(* IEC 61131-3 sources: zd/料盘/多料盘, 22 files *)

(* ---- E_料盘运动状态.st ---- *)
{attribute 'qualified_only'}
{attribute 'strict'}
TYPE E_料盘运动状态 :
(

	到取料位中 := 0,
	到放料位中 := 1,
	待机:=4,
	错误:=5,
	暂停:=6,
	手动定位中:=7,
	定位号定位中:=8,
	到初始位中:=9,
	指定取料中:=10,
	指定放料中:=11,
	手动取料中:=12,
	手动放料中:=13
);
END_TYPE

(* ---- S_多料盘管理数据.st ---- *)
TYPE S_多料盘管理数据 :
STRUCT
	料盘管理数据	:ARRAY[0..gvl_常量.最大料盘数量-1] OF S_料盘管理数据;
END_STRUCT
END_TYPE

(* ---- S_多料盘管理数据_HMI.st ---- *)
TYPE S_多料盘管理数据_HMI :
STRUCT
	料盘管理数据索引 :UINT;
	料盘管理数据当前索引 :UINT;
	料盘管理数据	: S_料盘管理数据;
END_STRUCT
END_TYPE

(* ---- S_多料盘管理输入.st ---- *)
TYPE S_多料盘管理输入 :
STRUCT
	手自动:BOOL;

	暂停	:BOOL;
	复位	:BOOL;
	急停	:BOOL;
	报警清除:BOOL;
	//料盘管理输入	:ARRAY[0..gvl_常量.最大料盘数量-1] OF S_料盘管理输入;

	料盘选择	:UINT;
	目标点位 : S_点位行列坐标;                // 目标点位坐标

	设置料盘为满料 : BOOL;
	设置料盘为空料 : BOOL;
	设置点位状态信号 : BOOL;              // 设置点位状态信号
	设置状态 : E_点位状态;                // 设置的状态值

    取料 : BOOL;
	放料 : BOOL;

    定位:BOOL;
    定位号:UINT;

	到初始位:BOOL;

	取料完成:BOOL;
	放料完成:BOOL;
END_STRUCT
END_TYPE

(* ---- S_多料盘管理输入HMI.st ---- *)
TYPE S_多料盘管理输入HMI :
STRUCT

	急停	:BOOL;
	报警清除:BOOL;
	料盘选择	:UINT;
	目标点位 : S_点位行列坐标;                // 目标点位坐标

	设置料盘为满料 : BOOL;
	设置料盘为空料 : BOOL;
	定位到点位信号 : BOOL;
	设置点位状态信号 : BOOL;              // 设置点位状态信号
	设置状态 : E_点位状态;                // 设置的状态值
	定位:BOOL;
    定位号:INT;
	到初始位:BOOL;
END_STRUCT
END_TYPE

(* ---- S_多料盘管理输入HMI_xg_V1.st ---- *)
TYPE S_多料盘管理输入HMI_xg_V1 :
STRUCT

	指定取料	:BOOL;
	指定放料	:BOOL;
	取料	:BOOL;
	放料	:BOOL;

END_STRUCT
END_TYPE

(* ---- S_多料盘管理输出.st ---- *)
TYPE S_多料盘管理输出 :
STRUCT
	定位号定位到位:ARRAY[0..4] OF BOOL;

	初始位定位到位:BOOL;

	占位:DINT;

	到达定位位置:BOOL;

	复位完成:BOOL;
	暂停完成:BOOL;
	料盘运动状态:INT;

    (* 控制输出 *)
    移动X轴信号 : BOOL;                   // X轴移动控制信号
    移动Y轴信号 : BOOL;                   // Y轴移动控制信号
	移动Z轴信号 : BOOL;                   // Z轴移动控制信号
    目标X位置 : REAL;                     // 目标X坐标
    目标Y位置 : REAL;                     // 目标Y坐标
	目标Z位置 : REAL;                     // 目标Z坐标

	当前X位置 : REAL;                     // 目标X坐标
    当前Y位置 : REAL;                     // 目标Y坐标
	当前Z位置 : REAL;                     // 目标Z坐标

	当前X速度 : REAL;                     // 目标X坐标
    当前Y速度 : REAL;                     // 目标Y坐标
	当前Z速度 : REAL;                     // 目标Z坐标

    (* 错误信息 *)
	错误:BOOL;
    错误代码 : E_错误码;
    错误信息 : STRING(100);               // 错误描述

	料盘管理输出	:ARRAY[0..gvl_常量.最大料盘数量-1] OF S_料盘管理输出;
END_STRUCT
END_TYPE

(* ---- S_多料盘管理配置.st ---- *)
TYPE S_多料盘管理配置 :
STRUCT
	x索引	:INT:=0;
	y索引	:INT:=1;
	z索引	:INT:=2;

	x速度:REAL:=50;
	x加速度:REAL:=500;
	x减速度:REAL:=500;

	y速度:REAL:=50;
	y加速度:REAL:=500;
	y减速度:REAL:=500;

// 	xy插补速度:REAL:=50;
// 	xy插补加速度:REAL:=500;
// 	xy插补减速度:REAL:=500;

	z速度:REAL:=50;
	z加速度:REAL:=500;
	z减速度:REAL:=500;

	x定位位置	:ARRAY[0..gvl_常量.最大料盘位置号数量-1] OF REAL:=[10];
	y定位位置	:ARRAY[0..gvl_常量.最大料盘位置号数量-1] OF REAL:=[10];
	z定位位置	:ARRAY[0..gvl_常量.最大料盘位置号数量-1] OF REAL:=[10];

	x轴待料位	:REAL:=10;
	y轴待料位	:REAL:=10;
	z轴待料位	:REAL:=10;

END_STRUCT
END_TYPE

(* ---- S_多料盘管理配置_HMI.st ---- *)
TYPE S_多料盘管理配置_HMI :
STRUCT

	多料盘管理配置: S_多料盘管理配置;
	料盘配置索引:UINT;
	当前料盘配置索引:UINT;

	占位1:REAL;
	占位2:REAL;
	占位3:REAL;
	占位4:REAL;
	占位5:REAL;
	占位6:REAL;
	料盘配置	: S_料盘配置;

	占位14:REAL;
	占位15:REAL;
	占位16:REAL;
	料盘工艺配置:  S_料盘工艺配置;

	多料盘工艺配置:S_多料盘工艺配置;

END_STRUCT
END_TYPE

(* ---- FC_SEL.st ---- *)
//G：BOOL 类型选择条件
//IN0：G = TRUE 时的返回值
//IN1：G = false 时的返回值

FUNCTION FC_SEL : int
VAR_INPUT
	G:BOOL;
	IN1:INT;
	IN2:INT;
END_VAR
VAR
END_VAR

// --- BEGIN IMPLEMENTATION ---

IF G=TRUE THEN
	FC_SEL:=IN1;
	RETURN;
ELSE
	FC_SEL:=IN2;
	RETURN;
END_IF

(* ---- FC_方向判断.st ---- *)
FUNCTION FC_方向判断 : INT
VAR_IN_OUT
	i方向X      : INT;
    i方向Y      : INT;
END_VAR
VAR_INPUT
	f起始点X     : REAL;
    f起始点Y     : REAL;
    f参考点X    : REAL;
    f参考点Y    : REAL;
END_VAR
VAR
	f间距X     : REAL;
    f间距Y     : REAL;
END_VAR

// --- BEGIN IMPLEMENTATION ---

i方向X :=0;
i方向Y :=0;
// 参考点和起始点不能相同
IF f参考点X =f起始点X OR f参考点Y = f起始点Y THEN
	FC_方向判断 := 1;   // 参参考点和起始点不能相同
	RETURN;
END_IF;

// 计算实际与理论的差值
f间距X := f参考点X - f起始点X;
f间距Y := f参考点Y - f起始点Y;

// 判断X方向
i方向X := FC_SEL(f间距X > 0.0, 1, -1);

// 判断Y方向
i方向Y := FC_SEL(f间距Y > 0.0, 1, -1);

(* ---- FB_多料盘管理.st ---- *)
FUNCTION_BLOCK FB_多料盘管理
VAR_IN_OUT
	x轴:SM3_Basic.AXIS_REF_VIRTUAL_SM3;
	y轴:SM3_Basic.AXIS_REF_VIRTUAL_SM3;
	z轴:SM3_Basic.AXIS_REF_VIRTUAL_SM3;

	多料盘管理数据:S_多料盘管理数据;
	多料盘管理输出:S_多料盘管理输出;
	ST_料盘配置V1_xg_0:ARRAY[0..gvl_常量.最大料盘数量-1] OF ST_料盘配置V1_xg;

END_VAR
VAR_INPUT
	全局状态:E_系统运行状态;
	使能:BOOL;
	多料盘管理输入HMI:S_多料盘管理输入HMI;
	S_多料盘管理输入HMI_xg_V1_0:S_多料盘管理输入HMI_xg_V1;
	多料盘管理输入	:S_多料盘管理输入;

	x轴配置:Ax_配置;
	y轴配置:Ax_配置;
	z轴配置:Ax_配置;
	x轴输出:Basic_Lib.Ax_输出;
	y轴输出:Basic_Lib.Ax_输出;
	z轴输出:Basic_Lib.Ax_输出;

	多料盘管理配置:S_多料盘管理配置;
	料盘配置	:ARRAY[0..gvl_常量.最大料盘数量-1] OF S_料盘配置;
	料盘工艺配置	:ARRAY[0..gvl_常量.最大料盘数量-1] OF S_料盘工艺配置;
	多料盘工艺配置	: S_多料盘工艺配置;
	//料盘轴运动输出:S_料盘轴运动输出;
END_VAR
VAR_OUTPUT
	料盘轴运动输入:S_料盘轴运动输入;
	料盘轴运动输出:S_料盘轴运动输出;
	报错料盘:INT;
END_VAR
VAR
	CheckID:Basic_Lib.FB_CheckID;
	//FB_G代码插补_0:FB_G代码插补;
	MC_MoveAbsolute_0: MC_MoveAbsolute;
	MC_MoveAbsolute_1: MC_MoveAbsolute;
	MC_MoveAbsolute_2: MC_MoveAbsolute;
	MC_Move_ChangePosVel_Pul_2: Basic_Lib.MC_Move_ChangePosVel_Pul;
	MC_Stop_1: MC_Stop;
	MC_Stop_2: MC_Stop;
	MC_Stop_3: MC_Stop;
	MC_Reset_0:MC_Reset;
	MC_Reset_1:MC_Reset;
	MC_Reset_2:MC_Reset;

	x轴状态:MC_ReadStatus;
	y轴状态:MC_ReadStatus;
	z轴状态:MC_ReadStatus;
	SMC3_ReinitDrive_0:SMC3_ReinitDrive;
	SMC3_ReinitDrive_1:SMC3_ReinitDrive;
	SMC3_ReinitDrive_2:SMC3_ReinitDrive;

	清空多料盘管理输出:S_多料盘管理输出;

	使能上升沿:R_TRIG;
	设置料盘满料上升沿 :  R_TRIG;  // 设置料盘满料上升沿
	设置料盘空料上升沿 :  R_TRIG;  // 设置料盘空料上升沿
	急停上升沿:  R_TRIG;

	取料上升沿 :  R_TRIG;  // 设置料盘满料上升沿
	放料上升沿 :  R_TRIG;  // 设置料盘空料上升沿
	定位上升沿 :  Standard.R_TRIG;
	到初始位上升沿:Standard.R_TRIG;

	取料完成上升沿 :  R_TRIG;
	放料完成上升沿 :  R_TRIG;
	错误上升沿:R_TRIG;

	手动设置点位状态上升沿:  R_TRIG;
	手动定位点位上升沿:  R_TRIG;
	手动急停上升沿:  R_TRIG;
	手动定位上升沿 :  Standard.R_TRIG;

	手动指定取料上升沿:  R_TRIG;
	手动指定放料上升沿:  R_TRIG;
	手动取料上升沿:  R_TRIG;
	手动放料上升沿:  R_TRIG;

	暂停上升沿:  R_TRIG;
	复位上升沿:  R_TRIG;

	i: INT;
	row: INT;
	col: INT;
	取料流程: INT;
	j: INT;
	临时定位行号: INT;
	临时定位列号: INT;

	z轴定位到位:BOOL;
	放料流程: INT;
	手动定位流程: INT;
	插补定位完成: BOOL;

	定位流程: INT;
	手动定位流程1: INT;

	手动x目标位置:REAL;
	手动y目标位置:REAL;
	手动z目标位置:REAL;

	指定x目标位置:REAL;
	指定y目标位置:REAL;
	指定z目标位置:REAL;

	z轴在待料位:BOOL;

	x轴定位到位: BOOL;
	y轴定位到位: BOOL;
	流程运行状态: BOOL;
	动作控制变量状态: BOOL;
	流程可运行: BOOL;
	轴可运动: BOOL;
	料盘管理输入: INT;
	暂停取料流程: INT;
	暂停定位流程: INT;
	错误前取料流程: INT;
	错误前放料流程: INT;
	错误前定位流程: INT;

	x取料方向X:INT;
	x取料方向Y:INT;
	x放料方向X:INT;
	x放料方向Y:INT;

	i行起始:INT;
	i行结束:INT;
	i列起始:INT;
	i列结束:INT;
	i行递增:INT;
	i列递增:INT;
	指定取料流程: INT;
	指定放料流程: INT;
	手动料盘选择:INT;
	手动取料流程: INT;
	手动放料流程: INT;
END_VAR

// --- BEGIN IMPLEMENTATION ---

(*========================输入控制========================*)
CheckID(xID检测:= TRUE, xID正确=> );
//IF NOT CheckID.xID正确 THEN RETURN; END_IF

IF ADR(x轴) = SM3_Basic.NULL THEN
    RETURN;
END_IF
IF ADR(y轴) = SM3_Basic.NULL  THEN
    RETURN;
END_IF
IF ADR(z轴) = SM3_Basic.NULL  THEN
    RETURN;
END_IF

使能上升沿(CLK:=使能 , Q=> );
IF NOT 使能 THEN
	放料流程:=0;
	取料流程:=0;
	定位流程:=0;
	手动定位流程:=0;
	指定取料流程:=0;
	指定放料流程:=0;
	手动取料流程:=0;
	手动放料流程:=0;
	多料盘管理输出.料盘运动状态:=E_料盘运动状态.待机;
	料盘轴运动输入.x轴定位:=FALSE;
	料盘轴运动输入.y轴定位:=FALSE;
	料盘轴运动输入.Z轴定位:=FALSE;
	料盘轴运动输入.插补启动:=FALSE;
	多料盘管理输出.错误:=FALSE;
	多料盘管理输出.错误信息:='';
	RETURN;
ELSE
	;
END_IF

ACT_自动状态控制();

设置料盘满料上升沿(CLK := (多料盘管理输入.设置料盘为满料  AND 多料盘管理输入.手自动) OR (多料盘管理输入HMI.设置料盘为满料  AND NOT 多料盘管理输入.手自动));
设置料盘空料上升沿(CLK := (多料盘管理输入.设置料盘为空料 AND 多料盘管理输入.手自动) OR (多料盘管理输入HMI.设置料盘为空料  AND NOT 多料盘管理输入.手自动));
(* 处理料盘设置满料信号 *)
IF 设置料盘满料上升沿.Q THEN
	(* 初始化指定料盘数据 *)
	FOR row := 0 TO GVL_常量.最大料盘行数 - 1 DO
		FOR col := 0 TO GVL_常量.最大料盘列数 - 1 DO
			IF 多料盘管理输入.料盘选择<=GVL_常量.最大料盘数量-1 THEN
				IF  多料盘管理输入.手自动 THEN
					多料盘管理数据.料盘管理数据[多料盘管理输入.料盘选择].点位状态[row, col] := E_点位状态.有料;
					多料盘管理数据.料盘管理数据[多料盘管理输入.料盘选择].屏蔽点位[row, col] := FALSE;
				ELSE
					多料盘管理数据.料盘管理数据[多料盘管理输入HMI.料盘选择].点位状态[row, col] := E_点位状态.有料;
					多料盘管理数据.料盘管理数据[多料盘管理输入HMI.料盘选择].屏蔽点位[row, col] := FALSE;
				END_IF

			END_IF

		END_FOR;
	END_FOR;
	IF 多料盘管理输入.料盘选择>GVL_常量.最大料盘数量-1 THEN
	FOR i := 0 TO GVL_常量.最大料盘数量 - 1 DO
		FOR row := 0 TO GVL_常量.最大料盘行数 - 1 DO
			FOR col := 0 TO GVL_常量.最大料盘列数 - 1 DO

				多料盘管理数据.料盘管理数据[i].点位状态[row, col] := E_点位状态.有料;
				多料盘管理数据.料盘管理数据[i].屏蔽点位[row, col] := FALSE;

			END_FOR;
		END_FOR;
	END_FOR
	END_IF
END_IF;

(* 处理料盘设置空料信号 *)
IF 设置料盘空料上升沿.Q THEN
	(* 初始化指定料盘数据 *)
	FOR row := 0 TO GVL_常量.最大料盘行数 - 1 DO
		FOR col := 0 TO GVL_常量.最大料盘列数 - 1 DO
			IF 多料盘管理输入.料盘选择<=GVL_常量.最大料盘数量-1 THEN
				IF  多料盘管理输入.手自动 THEN
					多料盘管理数据.料盘管理数据[多料盘管理输入.料盘选择].点位状态[row, col] := E_点位状态.无料;
					多料盘管理数据.料盘管理数据[多料盘管理输入.料盘选择].屏蔽点位[row, col] := FALSE;
				ELSE
					多料盘管理数据.料盘管理数据[多料盘管理输入HMI.料盘选择].点位状态[row, col] := E_点位状态.无料;
					多料盘管理数据.料盘管理数据[多料盘管理输入HMI.料盘选择].屏蔽点位[row, col] := FALSE;
				END_IF
			END_IF
		END_FOR;

		IF 多料盘管理输入.料盘选择>GVL_常量.最大料盘数量-1 THEN
		FOR i := 0 TO GVL_常量.最大料盘数量 - 1 DO
			FOR row := 0 TO GVL_常量.最大料盘行数 - 1 DO
				FOR col := 0 TO GVL_常量.最大料盘列数 - 1 DO

					多料盘管理数据.料盘管理数据[i].点位状态[row, col] := E_点位状态.无料;
					多料盘管理数据.料盘管理数据[i].屏蔽点位[row, col] := FALSE;

				END_FOR;
			END_FOR;
		END_FOR
		END_IF
	END_FOR;
END_IF;

手动设置点位状态上升沿(CLK:=多料盘管理输入HMI.设置点位状态信号 , Q=> );
IF 手动设置点位状态上升沿.Q AND ((多料盘管理输入HMI.目标点位.行号<>临时定位行号 OR 多料盘管理输入HMI.目标点位.列号<>临时定位列号)OR (放料流程=0 AND 取料流程=0))  THEN
	多料盘管理数据.料盘管理数据[多料盘管理输入HMI.料盘选择].点位状态[多料盘管理输入HMI.目标点位.行号,多料盘管理输入HMI.目标点位.列号]:=多料盘管理输入HMI.设置状态;
	多料盘管理数据.料盘管理数据[多料盘管理输入HMI.料盘选择].屏蔽点位[多料盘管理输入HMI.目标点位.行号,多料盘管理输入HMI.目标点位.列号]:=(多料盘管理输入HMI.设置状态=E_点位状态.屏蔽);
END_IF

流程可运行:=放料流程=0 AND 取料流程=0 AND 定位流程=0 AND 手动定位流程=0 AND 指定取料流程=0 AND 指定放料流程=0 AND 手动取料流程=0 AND 手动放料流程=0 ;

轴可运动:= x轴状态.Standstill AND y轴状态.Standstill AND z轴状态.Standstill ;
//x轴输出.x回零完成 AND y轴输出.x回零完成 AND z轴输出.x回零完成  AND

ACT_手动();
ACT_手动指定放料();
ACT_手动指定取料();
ACT_手动放料();
ACT_手动取料();
ACT_自动取料();
ACT_自动放料();
ACT_定位号插补();

ACT_FB();

多料盘管理输出.初始位定位到位:=(x轴.fActPosition<=(多料盘管理配置.x轴待料位+x轴配置.f到位偏差)) AND (x轴.fActPosition>=(多料盘管理配置.x轴待料位-x轴配置.f到位偏差))
	AND(y轴.fActPosition<=(多料盘管理配置.y轴待料位+y轴配置.f到位偏差)) AND (y轴.fActPosition>=(多料盘管理配置.y轴待料位-y轴配置.f到位偏差))
	AND (z轴.fActPosition<=(多料盘管理配置.z轴待料位+z轴配置.f到位偏差)) AND (z轴.fActPosition>=(多料盘管理配置.z轴待料位-z轴配置.f到位偏差)
	AND  x轴状态.Standstill AND y轴状态.Standstill AND z轴状态.Standstill );

插补定位完成:=((x轴.fActPosition<=(料盘轴运动输入.目标位置[0]+x轴配置.f到位偏差)) AND (x轴.fActPosition>=(料盘轴运动输入.目标位置[0]-x轴配置.f到位偏差))
AND(y轴.fActPosition<=(料盘轴运动输入.目标位置[1]+y轴配置.f到位偏差)) AND (y轴.fActPosition>=(料盘轴运动输入.目标位置[1]-y轴配置.f到位偏差)));

x轴定位到位:=((x轴.fActPosition<=(料盘轴运动输入.x定位位置+x轴配置.f到位偏差)) AND (x轴.fActPosition>=(料盘轴运动输入.x定位位置-x轴配置.f到位偏差)));
y轴定位到位:=((y轴.fActPosition<=(料盘轴运动输入.y定位位置+y轴配置.f到位偏差)) AND (y轴.fActPosition>=(料盘轴运动输入.y定位位置-y轴配置.f到位偏差)));
z轴定位到位:=((z轴.fActPosition<=(料盘轴运动输入.z定位位置+z轴配置.f到位偏差)) AND (z轴.fActPosition>=(料盘轴运动输入.z定位位置-z轴配置.f到位偏差)));

z轴在待料位:=(z轴.fActPosition<=(多料盘管理配置.z轴待料位+z轴配置.f到位偏差)) AND (z轴.fActPosition>=(多料盘管理配置.z轴待料位-z轴配置.f到位偏差));

ACT_料盘状态();

//手自动报警清除
IF 多料盘管理输入.报警清除 OR 多料盘管理输入hmi.报警清除 THEN
	多料盘管理输出.错误:=FALSE;
    多料盘管理输出.错误信息 :='';              // 系统错误描述
	//多料盘管理输出.料盘运动状态:=E_料盘运动状态.待机;
END_IF

IF 料盘轴运动输出.x定位错误 THEN 多料盘管理输出.错误:=TRUE; 多料盘管理输出.错误信息 := Standard.CONCAT('SMC_ERROR: ', TO_STRING(料盘轴运动输出.x定位错误码));多料盘管理输出.错误代码:=E_错误码.料盘X轴定位错误; END_IF
IF 料盘轴运动输出.y定位错误 THEN 多料盘管理输出.错误:=TRUE; 多料盘管理输出.错误信息 := Standard.CONCAT('SMC_ERROR: ', TO_STRING(料盘轴运动输出.y定位错误码));多料盘管理输出.错误代码:=E_错误码.料盘Y轴定位错误; END_IF
IF 料盘轴运动输出.z定位错误 THEN 多料盘管理输出.错误:=TRUE; 多料盘管理输出.错误信息 :=MC_Move_ChangePosVel_Pul_2.s错误码; (*Standard.CONCAT('SMC_ERROR: ', TO_STRING(料盘轴运动输出.z定位错误码));*)多料盘管理输出.错误代码:=E_错误码.料盘Z轴定位错误; END_IF
//IF LS_2AxisLine_1.Error  THEN 多料盘管理输出.错误:=TRUE; 多料盘管理输出.错误信息 := Standard.CONCAT('SMC_ERROR: ', TO_STRING(LS_2AxisLine_1.ErrorID)); 多料盘管理输出.错误代码:=3; END_IF
//IF 料盘轴运动输出.插补错误 THEN 多料盘管理输出.错误:=TRUE; 多料盘管理输出.错误信息 := 料盘轴运动输出.插补错误码;多料盘管理输出.错误代码:=3; END_IF

错误上升沿(CLK:= 多料盘管理输出.错误, Q=> );
IF 错误上升沿.Q THEN
	;
	放料流程:=0;
	取料流程:=0;
	定位流程:=0;
	手动定位流程:=0;
	指定取料流程:=0;
	指定放料流程:=0;
	手动取料流程:=0;
	手动放料流程:=0;
	料盘轴运动输入.x轴定位:=FALSE;
	料盘轴运动输入.y轴定位:=FALSE;
	料盘轴运动输入.Z轴定位:=FALSE;
	料盘轴运动输入.插补启动:=FALSE;
	多料盘管理输出.料盘运动状态:=E_料盘运动状态.错误;
END_IF

IF 多料盘管理输出.错误 THEN
	;
	放料流程:=0;
	取料流程:=0;
	定位流程:=0;
	手动定位流程:=0;
	指定取料流程:=0;
	手动取料流程:=0;
	手动放料流程:=0;
	料盘轴运动输入.x轴定位:=FALSE;
	料盘轴运动输入.y轴定位:=FALSE;
	料盘轴运动输入.Z轴定位:=FALSE;
	料盘轴运动输入.插补启动:=FALSE;
END_IF

(* ---- FB_多料盘管理.ACT_定位号插补.action.st ---- *)
定位上升沿(CLK:=多料盘管理输入.定位 AND 多料盘管理输入.手自动 , Q=> );

IF GVL_系统变量.全局状态=E_系统运行状态.系统状态_故障 THEN
	料盘轴运动输入.x轴定位:=FALSE;
	料盘轴运动输入.y轴定位:=FALSE;
	料盘轴运动输入.Z轴定位:=FALSE;
	料盘轴运动输入.插补启动:=FALSE;
	RETURN;
END_IF

IF GVL_系统变量.全局状态<>E_系统运行状态.系统状态_运行 AND GVL_系统变量.全局状态<>E_系统运行状态.系统状态_清料中  AND GVL_系统变量.全局状态<>E_系统运行状态.系统状态_暂停中 THEN

	RETURN;
END_IF
IF 定位上升沿.Q AND 轴可运动 AND 流程可运行
	AND NOT 多料盘管理输入.到初始位 AND NOT 多料盘管理输入.取料 AND NOT 多料盘管理输入.放料
	 AND NOT 多料盘管理输入.暂停 AND NOT 多料盘管理输出.错误
	AND 多料盘管理输入.定位号>=0 AND 多料盘管理输入.定位号<5 AND

	(多料盘管理输出.料盘运动状态=E_料盘运动状态.待机
	OR 多料盘管理输出.料盘运动状态=E_料盘运动状态.暂停)
THEN

		料盘轴运动输入.x轴定位:=FALSE;
		料盘轴运动输入.y轴定位:=FALSE;
		料盘轴运动输入.Z轴定位:=FALSE;
		料盘轴运动输入.插补启动:=FALSE;
		多料盘管理输出.定位号定位到位[多料盘管理输入.定位号]:=FALSE;
		多料盘管理输出.料盘运动状态:=E_料盘运动状态.定位号定位中;
		定位流程:=2;

ELSE
	;
END_IF;

IF 定位流程=2 THEN
	IF z轴在待料位=FALSE AND NOT 多料盘管理输入.暂停 THEN
		料盘轴运动输入.z定位位置:=多料盘管理输出.目标Z位置 := 多料盘管理配置.z轴待料位;
		料盘轴运动输入.z定位速度:=多料盘管理配置.z速度;
		料盘轴运动输入.z定位加速度:=多料盘管理配置.z加速度;
		料盘轴运动输入.z定位减速度:=多料盘管理配置.z减速度;
		(* 移动轴 *)
		多料盘管理输出.移动Z轴信号 := TRUE;
		料盘轴运动输入.Z轴定位:=TRUE;
	ELSIF z轴在待料位 AND NOT 多料盘管理输入.暂停 THEN
		多料盘管理输出.移动Z轴信号 := FALSE;
		料盘轴运动输入.Z轴定位:=FALSE;
		定位流程:=5;
	ELSIF  多料盘管理输入.暂停 THEN
		多料盘管理输出.暂停完成:=TRUE;
	END_IF
END_IF

IF 定位流程=5 THEN

		多料盘管理输出.移动X轴信号 := FALSE;
		多料盘管理输出.移动Y轴信号 := FALSE;

		//料盘轴运动输入.插补启动:=FALSE;

		料盘轴运动输入.x轴定位:=FALSE;
		料盘轴运动输入.y轴定位:=FALSE;
		料盘轴运动输入.x定位位置:=料盘轴运动输入.目标位置[0] :=多料盘管理输出.目标X位置 := 多料盘管理配置.x定位位置[多料盘管理输入.定位号];

		料盘轴运动输入.y定位位置:=料盘轴运动输入.目标位置[1] :=多料盘管理输出.目标Y位置 := 多料盘管理配置.y定位位置[多料盘管理输入.定位号];

		料盘轴运动输入.z定位位置:=多料盘管理输出.目标Z位置 := 多料盘管理配置.z定位位置[多料盘管理输入.定位号];
		// 		料盘轴运动输入.xy插补速度:=多料盘管理配置.xy插补速度;
		// 		料盘轴运动输入.xy插补加速度:=多料盘管理配置.xy插补加速度;
		// 		料盘轴运动输入.xy插补减速度:=多料盘管理配置.xy插补减速度;
		料盘轴运动输入.x定位速度:=多料盘管理配置.x速度;
		料盘轴运动输入.x定位加速度:=多料盘管理配置.x加速度;
		料盘轴运动输入.x定位减速度:=多料盘管理配置.x减速度;

		料盘轴运动输入.y定位速度:=多料盘管理配置.y速度;
		料盘轴运动输入.y定位加速度:=多料盘管理配置.y加速度;
		料盘轴运动输入.y定位减速度:=多料盘管理配置.y减速度;

		IF 多料盘工艺配置.位置号z轴下降减速[多料盘管理输入.定位号].启用=1 THEN
			IF z轴.fActPosition>多料盘工艺配置.位置号z轴下降减速[多料盘管理输入.定位号].z定位减速位置 THEN
				料盘轴运动输入.z定位速度:= 多料盘工艺配置.位置号z轴下降减速[多料盘管理输入.定位号].z定位减速速度;
			ELSE
				料盘轴运动输入.z定位速度:=多料盘管理配置.z速度;
			END_IF
		ELSE
			料盘轴运动输入.z定位速度:=多料盘管理配置.z速度;
		END_IF
		料盘轴运动输入.z定位速度:=多料盘管理配置.z速度;
		料盘轴运动输入.z定位加速度:=多料盘管理配置.z加速度;
		料盘轴运动输入.z定位减速度:=多料盘管理配置.z减速度;

		定位流程:=10;

ELSIF 定位流程=10 THEN

	(* 移动轴 *)

	IF 插补定位完成=FALSE AND x轴.nAxisState=Standstill  AND y轴.nAxisState=Standstill AND NOT 多料盘管理输入.暂停 THEN
		多料盘管理输出.移动X轴信号 := TRUE;
		多料盘管理输出.移动Y轴信号 := TRUE;
		//料盘轴运动输入.插补启动:=TRUE;
		料盘轴运动输入.x轴定位:=TRUE;
		料盘轴运动输入.y轴定位:=TRUE;
	ELSIF 插补定位完成 AND x轴.nAxisState=Standstill  AND y轴.nAxisState=Standstill AND NOT 多料盘管理输入.暂停 THEN
		多料盘管理输出.移动X轴信号 := FALSE;
		多料盘管理输出.移动Y轴信号 := FALSE;

		//料盘轴运动输入.插补启动:=FALSE;

		料盘轴运动输入.x轴定位:=FALSE;
		料盘轴运动输入.y轴定位:=FALSE;
		定位流程:=12;
	ELSIF  多料盘管理输入.暂停 THEN
		多料盘管理输出.暂停完成:=TRUE;
	END_IF
ELSIF 定位流程=12 THEN

		IF 多料盘工艺配置.位置号z轴下降减速[多料盘管理输入.定位号].启用=1 THEN
			IF z轴.fActPosition>多料盘工艺配置.位置号z轴下降减速[多料盘管理输入.定位号].z定位减速位置 THEN
				料盘轴运动输入.z定位速度:= 多料盘工艺配置.位置号z轴下降减速[多料盘管理输入.定位号].z定位减速速度;
			END_IF
		END_IF
		IF z轴定位到位=FALSE AND  z轴.nAxisState=Standstill  AND NOT 多料盘管理输入.暂停 THEN
			(* 移动轴 *)
			多料盘管理输出.移动Z轴信号 := TRUE;
			料盘轴运动输入.Z轴定位:=TRUE;
		ELSIF z轴定位到位 AND z轴.nAxisState=Standstill AND NOT 多料盘管理输入.暂停 THEN
			多料盘管理输出.移动Z轴信号 := FALSE;
			料盘轴运动输入.Z轴定位:=FALSE;
			定位流程:=13;
		ELSIF z轴定位到位 AND 多料盘管理输入.暂停 THEN
			多料盘管理输出.暂停完成:=TRUE;
		END_IF

END_IF

IF 定位流程=13 THEN

		IF 多料盘管理输出.料盘运动状态=E_料盘运动状态.定位号定位中 THEN
			IF 多料盘工艺配置.位置号附加动作[多料盘管理输入.定位号].位置号附加动作=0 THEN
				多料盘管理输出.料盘运动状态:=E_料盘运动状态.待机;
				多料盘管理输出.定位号定位到位[多料盘管理输入.定位号]:=TRUE;
				定位流程:=0;
			ELSIF 多料盘工艺配置.位置号附加动作[多料盘管理输入.定位号].位置号附加动作=1 THEN
				定位流程:=20;
			END_IF
		ELSE
			多料盘管理输出.料盘运动状态:=E_料盘运动状态.待机;
			定位流程:=0;
		END_IF

ELSIF 定位流程=20 THEN
	IF 多料盘工艺配置.位置号附加动作[多料盘管理输入.定位号].索引=0 AND x轴.nAxisState=Standstill AND NOT 多料盘管理输入.暂停 THEN
		料盘轴运动输入.X定位位置:=多料盘管理输出.目标X位置 := 多料盘工艺配置.位置号附加动作[多料盘管理输入.定位号].偏移值+x轴.fActPosition;
		料盘轴运动输入.x定位速度:= 多料盘工艺配置.位置号附加动作[多料盘管理输入.定位号].速度;
		料盘轴运动输入.x定位加速度:= 多料盘工艺配置.位置号附加动作[多料盘管理输入.定位号].加速度;
		料盘轴运动输入.x定位减速度:=多料盘工艺配置.位置号附加动作[多料盘管理输入.定位号].减速度;
		多料盘管理输出.移动X轴信号 := TRUE;
		料盘轴运动输入.x轴定位:=TRUE;
		定位流程:=30;
	ELSIF 多料盘工艺配置.位置号附加动作[多料盘管理输入.定位号].索引=1 AND y轴.nAxisState=Standstill AND NOT 多料盘管理输入.暂停 THEN
		料盘轴运动输入.y定位位置:=多料盘管理输出.目标y位置 := 多料盘工艺配置.位置号附加动作[多料盘管理输入.定位号].偏移值+y轴.fActPosition;
		料盘轴运动输入.y定位速度:=多料盘工艺配置.位置号附加动作[多料盘管理输入.定位号].速度;
		料盘轴运动输入.y定位加速度:=多料盘工艺配置.位置号附加动作[多料盘管理输入.定位号].加速度;
		料盘轴运动输入.y定位减速度:=多料盘工艺配置.位置号附加动作[多料盘管理输入.定位号].减速度;
		多料盘管理输出.移动y轴信号 := TRUE;
		料盘轴运动输入.y轴定位:=TRUE;
		定位流程:=30;
	ELSIF 多料盘工艺配置.位置号附加动作[多料盘管理输入.定位号].索引=2 AND z轴.nAxisState=Standstill AND NOT 多料盘管理输入.暂停 THEN
		料盘轴运动输入.z定位位置:=多料盘管理输出.目标z位置 := 多料盘工艺配置.位置号附加动作[多料盘管理输入.定位号].偏移值+z轴.fActPosition;
		料盘轴运动输入.z定位速度:=多料盘工艺配置.位置号附加动作[多料盘管理输入.定位号].速度;
		料盘轴运动输入.z定位加速度:=多料盘工艺配置.位置号附加动作[多料盘管理输入.定位号].加速度;
		料盘轴运动输入.z定位减速度:=多料盘工艺配置.位置号附加动作[多料盘管理输入.定位号].减速度;
		多料盘管理输出.移动z轴信号 := TRUE;
		料盘轴运动输入.z轴定位:=TRUE;
		定位流程:=30;
	ELSIF 多料盘管理输入.暂停 THEN
		多料盘管理输出.暂停完成:=TRUE;
	END_IF

ELSIF 定位流程=30 THEN
	IF 多料盘工艺配置.位置号附加动作[多料盘管理输入.定位号].索引=0 THEN
		IF x轴定位到位 AND x轴.nAxisState=Standstill THEN
			料盘轴运动输入.x轴定位:=FALSE;
			多料盘管理输出.移动X轴信号 := FALSE;
			多料盘管理输出.料盘运动状态:=E_料盘运动状态.待机;
			多料盘管理输出.定位号定位到位[多料盘管理输入.定位号]:=TRUE;
			定位流程:=0;
		END_IF
	ELSIF 多料盘工艺配置.位置号附加动作[多料盘管理输入.定位号].索引=1 THEN
		IF y轴定位到位 AND y轴.nAxisState=Standstill THEN
			料盘轴运动输入.y轴定位:=FALSE;
			多料盘管理输出.移动y轴信号 := FALSE;
			多料盘管理输出.料盘运动状态:=E_料盘运动状态.待机;
			多料盘管理输出.定位号定位到位[多料盘管理输入.定位号]:=TRUE;
			定位流程:=0;
		END_IF
	ELSIF 多料盘工艺配置.位置号附加动作[多料盘管理输入.定位号].索引=2 THEN
		IF z轴定位到位 AND z轴.nAxisState=Standstill THEN
			料盘轴运动输入.z轴定位:=FALSE;
			多料盘管理输出.移动z轴信号 := FALSE;
			多料盘管理输出.料盘运动状态:=E_料盘运动状态.待机;
			多料盘管理输出.定位号定位到位[多料盘管理输入.定位号]:=TRUE;
			定位流程:=0;
		END_IF
	END_IF
END_IF

(* ---- FB_多料盘管理.ACT_手动.action.st ---- *)
手动定位上升沿(CLK:=多料盘管理输入HMI.定位 AND NOT 多料盘管理输入.手自动, Q=> );
到初始位上升沿(CLK:=多料盘管理输入HMI.到初始位 AND NOT 多料盘管理输入.手自动  , Q=> );
手动定位点位上升沿(CLK:=多料盘管理输入HMI.定位到点位信号 AND NOT 多料盘管理输入.手自动 , Q=> );

IF 手动定位点位上升沿.Q AND 轴可运动 AND 流程可运行 THEN
	料盘轴运动输入.x轴定位:=FALSE;
	料盘轴运动输入.y轴定位:=FALSE;
	料盘轴运动输入.Z轴定位:=FALSE;
	料盘轴运动输入.插补启动:=FALSE;
	手动定位流程:=2;
	多料盘管理输出.料盘运动状态:=E_料盘运动状态.手动定位中;

END_IF

IF 手动定位上升沿.Q AND 轴可运动 AND 流程可运行  THEN
	料盘轴运动输入.x轴定位:=FALSE;
	料盘轴运动输入.y轴定位:=FALSE;
	料盘轴运动输入.Z轴定位:=FALSE;
	料盘轴运动输入.插补启动:=FALSE;
	多料盘管理输出.定位号定位到位[多料盘管理输入hmi.定位号]:=FALSE;
	手动定位流程:=2;
	多料盘管理输出.料盘运动状态:=E_料盘运动状态.定位号定位中;

END_IF

IF 到初始位上升沿.Q  AND 轴可运动 AND 流程可运行 THEN
	料盘轴运动输入.x轴定位:=FALSE;
	料盘轴运动输入.y轴定位:=FALSE;
	料盘轴运动输入.Z轴定位:=FALSE;
	料盘轴运动输入.插补启动:=FALSE;
	多料盘管理输出.料盘运动状态:=E_料盘运动状态.到初始位中;
	手动定位流程:=2;

ELSE
	;
END_IF;

手动x目标位置:=料盘配置[多料盘管理输入HMI.料盘选择].起始X坐标 +
								多料盘管理输入HMI.目标点位.列号 * 料盘配置[多料盘管理输入HMI.料盘选择].列间距 +
								料盘配置[多料盘管理输入HMI.料盘选择].点位偏移[多料盘管理输入HMI.目标点位.行号, 多料盘管理输入HMI.目标点位.列号].x点位偏移;
手动y目标位置:=	料盘配置[多料盘管理输入HMI.料盘选择].起始Y坐标 +
								多料盘管理输入HMI.目标点位.行号 * 料盘配置[多料盘管理输入HMI.料盘选择].行间距 +
								料盘配置[多料盘管理输入HMI.料盘选择].点位偏移[多料盘管理输入HMI.目标点位.行号, 多料盘管理输入HMI.目标点位.列号].y点位偏移;
手动z目标位置:=料盘配置[多料盘管理输入HMI.料盘选择].Z轴高度 +
								料盘配置[多料盘管理输入HMI.料盘选择].点位偏移[多料盘管理输入HMI.目标点位.行号, 多料盘管理输入HMI.目标点位.列号].z点位偏移;

IF 手动定位流程=2 THEN
	IF z轴在待料位=FALSE THEN
		料盘轴运动输入.z定位位置:=多料盘管理输出.目标Z位置 := 多料盘管理配置.z轴待料位;
		料盘轴运动输入.z定位速度:=多料盘管理配置.z速度;
		料盘轴运动输入.z定位加速度:=多料盘管理配置.z加速度;
		料盘轴运动输入.z定位减速度:=多料盘管理配置.z减速度;
		料盘轴运动输入.Z轴定位:=TRUE;
		手动定位流程:=5;
	ELSE
		手动定位流程:=5;
	END_IF
END_IF

IF 手动定位流程=5 THEN
	IF z轴在待料位 AND z轴.nAxisState=Standstill  THEN
		IF 多料盘管理输出.料盘运动状态=E_料盘运动状态.手动定位中 THEN
			料盘轴运动输入.x定位位置:=料盘轴运动输入.目标位置[0] :=多料盘管理输出.目标X位置 := 料盘配置[多料盘管理输入HMI.料盘选择].起始X坐标 +
									多料盘管理输入HMI.目标点位.列号 * 料盘配置[多料盘管理输入HMI.料盘选择].列间距 +
									料盘配置[多料盘管理输入HMI.料盘选择].点位偏移[多料盘管理输入HMI.目标点位.行号, 多料盘管理输入HMI.目标点位.列号].x点位偏移;

			料盘轴运动输入.y定位位置:=料盘轴运动输入.目标位置[1] :=多料盘管理输出.目标Y位置 := 料盘配置[多料盘管理输入HMI.料盘选择].起始Y坐标 +
										多料盘管理输入HMI.目标点位.行号 * 料盘配置[多料盘管理输入HMI.料盘选择].行间距 +
										料盘配置[多料盘管理输入HMI.料盘选择].点位偏移[多料盘管理输入HMI.目标点位.行号, 多料盘管理输入HMI.目标点位.列号].y点位偏移;

			料盘轴运动输入.z定位位置:=多料盘管理输出.目标Z位置 := 料盘配置[多料盘管理输入HMI.料盘选择].Z轴高度 +
										料盘配置[多料盘管理输入HMI.料盘选择].点位偏移[多料盘管理输入HMI.目标点位.行号, 多料盘管理输入HMI.目标点位.列号].z点位偏移;
		ELSIF 多料盘管理输出.料盘运动状态=E_料盘运动状态.定位号定位中 THEN
			料盘轴运动输入.x定位位置:=料盘轴运动输入.目标位置[0] :=多料盘管理输出.目标X位置 := 多料盘管理配置.x定位位置[多料盘管理输入HMI.定位号];

			料盘轴运动输入.y定位位置:=料盘轴运动输入.目标位置[1] :=多料盘管理输出.目标Y位置 := 多料盘管理配置.y定位位置[多料盘管理输入HMI.定位号];

			料盘轴运动输入.z定位位置:=多料盘管理输出.目标Z位置 := 多料盘管理配置.z定位位置[多料盘管理输入HMI.定位号];
		ELSIF 多料盘管理输出.料盘运动状态=E_料盘运动状态.到初始位中 THEN
			料盘轴运动输入.x定位位置:=料盘轴运动输入.目标位置[0] :=多料盘管理输出.目标X位置 := 多料盘管理配置.x轴待料位;

			料盘轴运动输入.y定位位置:=料盘轴运动输入.目标位置[1] :=多料盘管理输出.目标Y位置 := 多料盘管理配置.y轴待料位;

			料盘轴运动输入.z定位位置:=多料盘管理输出.目标Z位置 := 多料盘管理配置.z轴待料位;
		END_IF
// 		料盘轴运动输入.xy插补速度:=多料盘管理配置.xy插补速度;
// 		料盘轴运动输入.xy插补加速度:=多料盘管理配置.xy插补加速度;
// 		料盘轴运动输入.xy插补减速度:=多料盘管理配置.xy插补减速度;

		料盘轴运动输入.x定位速度:=多料盘管理配置.x速度;
		料盘轴运动输入.x定位加速度:=多料盘管理配置.x加速度;
		料盘轴运动输入.x定位减速度:=多料盘管理配置.x减速度;

		料盘轴运动输入.y定位速度:=多料盘管理配置.y速度;
		料盘轴运动输入.y定位加速度:=多料盘管理配置.y加速度;
		料盘轴运动输入.y定位减速度:=多料盘管理配置.y减速度;

		料盘轴运动输入.z定位速度:=多料盘管理配置.z速度;
		料盘轴运动输入.z定位加速度:=多料盘管理配置.z加速度;
		料盘轴运动输入.z定位减速度:=多料盘管理配置.z减速度;
		料盘轴运动输入.Z轴定位:=FALSE;
		手动定位流程:=10;

	END_IF
END_IF

IF 手动定位流程=10 THEN

	//料盘轴运动输入.插补启动:=TRUE;

	料盘轴运动输入.x轴定位:=TRUE;
	料盘轴运动输入.y轴定位:=TRUE;

	手动定位流程:=12;
ELSIF 手动定位流程=12 THEN
	IF 插补定位完成 AND x轴.nAxisState=Standstill  AND y轴.nAxisState=Standstill  THEN

		//料盘轴运动输入.插补启动:=FALSE;

		料盘轴运动输入.x轴定位:=FALSE;
		料盘轴运动输入.y轴定位:=FALSE;

		IF z轴.nAxisState=Standstill  THEN
			料盘轴运动输入.Z轴定位:=TRUE;
			手动定位流程:=13;
		END_IF

	END_IF
END_IF

IF 手动定位流程=13 THEN
	IF 多料盘管理输出.料盘运动状态=E_料盘运动状态.定位号定位中 THEN
		IF 多料盘工艺配置.位置号z轴下降减速[多料盘管理输入HMI.定位号].启用=1 THEN
			IF z轴.fActPosition>多料盘工艺配置.位置号z轴下降减速[多料盘管理输入HMI.定位号].z定位减速位置 THEN
				料盘轴运动输入.z定位速度:= 多料盘工艺配置.位置号z轴下降减速[多料盘管理输入HMI.定位号].z定位减速速度;		END_IF
		END_IF
	END_IF
	IF z轴定位到位 AND z轴.nAxisState=Standstill  THEN
		料盘轴运动输入.Z轴定位:=FALSE;
		IF 多料盘管理输出.料盘运动状态=E_料盘运动状态.定位号定位中 THEN
			IF 多料盘工艺配置.位置号附加动作[多料盘管理输入hmi.定位号].位置号附加动作=0 THEN
				多料盘管理输出.料盘运动状态:=E_料盘运动状态.待机;
				多料盘管理输出.定位号定位到位[多料盘管理输入hmi.定位号]:=TRUE;
				手动定位流程:=0;
			ELSIF 多料盘工艺配置.位置号附加动作[多料盘管理输入hmi.定位号].位置号附加动作=1 THEN
				手动定位流程:=20;
			END_IF
		ELSE
			多料盘管理输出.料盘运动状态:=E_料盘运动状态.待机;
			手动定位流程:=0;
		END_IF

	END_IF

ELSIF 手动定位流程=20 THEN
	IF 多料盘工艺配置.位置号附加动作[多料盘管理输入hmi.定位号].索引=0 THEN
		料盘轴运动输入.X定位位置:=多料盘管理输出.目标X位置 := 多料盘工艺配置.位置号附加动作[多料盘管理输入hmi.定位号].偏移值+x轴.fActPosition;
		料盘轴运动输入.x定位速度:= 多料盘工艺配置.位置号附加动作[多料盘管理输入hmi.定位号].速度;
		料盘轴运动输入.x定位加速度:= 多料盘工艺配置.位置号附加动作[多料盘管理输入hmi.定位号].加速度;
		料盘轴运动输入.x定位减速度:=多料盘工艺配置.位置号附加动作[多料盘管理输入hmi.定位号].减速度;
		料盘轴运动输入.x轴定位:=TRUE;
		手动定位流程:=30;
	ELSIF 多料盘工艺配置.位置号附加动作[多料盘管理输入hmi.定位号].索引=1 THEN
		料盘轴运动输入.y定位位置:=多料盘管理输出.目标y位置 := 多料盘工艺配置.位置号附加动作[多料盘管理输入hmi.定位号].偏移值+y轴.fActPosition;
		料盘轴运动输入.y定位速度:=多料盘工艺配置.位置号附加动作[多料盘管理输入hmi.定位号].速度;
		料盘轴运动输入.y定位加速度:=多料盘工艺配置.位置号附加动作[多料盘管理输入hmi.定位号].加速度;
		料盘轴运动输入.y定位减速度:=多料盘工艺配置.位置号附加动作[多料盘管理输入hmi.定位号].减速度;
		料盘轴运动输入.y轴定位:=TRUE;
		手动定位流程:=30;
	ELSIF 多料盘工艺配置.位置号附加动作[多料盘管理输入hmi.定位号].索引=2 THEN
		料盘轴运动输入.z定位位置:=多料盘管理输出.目标z位置 := 多料盘工艺配置.位置号附加动作[多料盘管理输入hmi.定位号].偏移值+z轴.fActPosition;
		料盘轴运动输入.z定位速度:=多料盘工艺配置.位置号附加动作[多料盘管理输入hmi.定位号].速度;
		料盘轴运动输入.z定位加速度:=多料盘工艺配置.位置号附加动作[多料盘管理输入hmi.定位号].加速度;
		料盘轴运动输入.z定位减速度:=多料盘工艺配置.位置号附加动作[多料盘管理输入hmi.定位号].减速度;
		料盘轴运动输入.z轴定位:=TRUE;
		手动定位流程:=30;
	END_IF

ELSIF 手动定位流程=30 THEN
	IF 多料盘工艺配置.位置号附加动作[多料盘管理输入hmi.定位号].索引=0 THEN
		IF x轴定位到位 AND x轴.nAxisState=Standstill  THEN
			料盘轴运动输入.x轴定位:=FALSE;
			多料盘管理输出.料盘运动状态:=E_料盘运动状态.待机;
			多料盘管理输出.定位号定位到位[多料盘管理输入hmi.定位号]:=TRUE;
			手动定位流程:=0;
		END_IF
	ELSIF 多料盘工艺配置.位置号附加动作[多料盘管理输入hmi.定位号].索引=1 THEN
		IF y轴定位到位 AND y轴.nAxisState=Standstill  THEN
			料盘轴运动输入.y轴定位:=FALSE;
			多料盘管理输出.料盘运动状态:=E_料盘运动状态.待机;
			多料盘管理输出.定位号定位到位[多料盘管理输入hmi.定位号]:=TRUE;
			手动定位流程:=0;
		END_IF
	ELSIF 多料盘工艺配置.位置号附加动作[多料盘管理输入hmi.定位号].索引=2 THEN
		IF z轴定位到位 AND z轴.nAxisState=Standstill  THEN
			料盘轴运动输入.z轴定位:=FALSE;
			多料盘管理输出.料盘运动状态:=E_料盘运动状态.待机;
			多料盘管理输出.定位号定位到位[多料盘管理输入hmi.定位号]:=TRUE;
			手动定位流程:=0;
		END_IF
	END_IF
END_IF

(* ---- FB_多料盘管理.ACT_手动取料.action.st ---- *)
手动取料上升沿(CLK:=S_多料盘管理输入HMI_xg_V1_0.取料 AND NOT 多料盘管理输入.手自动, Q=> );

IF 手动取料上升沿.Q AND 轴可运动 AND 流程可运行
THEN
	料盘轴运动输入.x轴定位:=FALSE;
	料盘轴运动输入.y轴定位:=FALSE;
	料盘轴运动输入.Z轴定位:=FALSE;
	料盘轴运动输入.插补启动:=FALSE;
	手动料盘选择:=多料盘管理输入hmi.料盘选择;
	手动取料流程:=2;
	多料盘管理输出.料盘运动状态:=E_料盘运动状态.手动取料中;

ELSE
	;
END_IF;

IF 手动取料流程=2 THEN
	IF z轴在待料位=FALSE THEN
		料盘轴运动输入.z定位位置:= 多料盘管理输出.目标Z位置 := 多料盘管理配置.z轴待料位;
		料盘轴运动输入.z定位速度:=多料盘管理配置.z速度;
		料盘轴运动输入.z定位加速度:=多料盘管理配置.z加速度;
		料盘轴运动输入.z定位减速度:=多料盘管理配置.z减速度;
		料盘轴运动输入.Z轴定位:=TRUE;
		手动取料流程:=5;
	ELSE
		手动取料流程:=5;
	END_IF
END_IF

IF 手动取料流程=5 THEN
	IF z轴在待料位=FALSE THEN
		料盘轴运动输入.z定位位置:= 多料盘管理输出.目标Z位置 := 多料盘管理配置.z轴待料位;
		料盘轴运动输入.z定位速度:=多料盘管理配置.z速度;
		料盘轴运动输入.z定位加速度:=多料盘管理配置.z加速度;
		料盘轴运动输入.z定位减速度:=多料盘管理配置.z减速度;
		料盘轴运动输入.Z轴定位:=TRUE;
	END_IF
	IF z轴在待料位 AND z轴.nAxisState=Standstill AND NOT 多料盘管理输入.暂停  THEN
		料盘轴运动输入.Z轴定位:=FALSE;
		手动取料流程:=6;
	ELSIF 多料盘管理输入.暂停 THEN
		多料盘管理输出.暂停完成:=TRUE;
	END_IF
END_IF

IF 手动取料流程=6 THEN
	IF FC_方向判断(
	i方向X:= x取料方向X,
	i方向Y:= x取料方向Y ,
	f起始点X:=料盘配置[手动料盘选择].起始X坐标 ,
	f起始点Y:= 料盘配置[手动料盘选择].起始Y坐标 ,
	f参考点X:=ST_料盘配置V1_xg_0[手动料盘选择].lf取料参考点x坐标 ,
	f参考点Y:=ST_料盘配置V1_xg_0[手动料盘选择].lf取料参考点y坐标 )=1 THEN
		多料盘管理输出.错误:=TRUE;
		报错料盘:=手动料盘选择;
		多料盘管理输出.错误信息 :=Standard.CONCAT(Standard.CONCAT('料盘', TO_STRING(手动料盘选择)), '取料参考点错误,不能和起始点相同');
		多料盘管理输出.错误代码:=E_错误码.取料参考点错误不能和起始点相同;
	ELSE
		手动取料流程:=7;
	END_IF
END_IF

IF 手动取料流程=7 THEN
	//左上
		IF ST_料盘配置V1_xg_0[手动料盘选择].x取料方位=0 THEN
			i行起始:=0;
			i行结束:=料盘配置[手动料盘选择].行数-1;
			i列起始:=0;
			i列结束:=料盘配置[手动料盘选择].列数-1;
			i行递增:=1;
			i列递增:=1;
		ELSIF ST_料盘配置V1_xg_0[手动料盘选择].x取料方位=1 THEN
			i行起始:=0;
			i行结束:=料盘配置[手动料盘选择].行数-1;
			i列起始:=料盘配置[手动料盘选择].列数-1;
			i列结束:=0;
			i行递增:=1;
			i列递增:=-1;
		ELSIF ST_料盘配置V1_xg_0[手动料盘选择].x取料方位=2 THEN
			i行起始:=料盘配置[手动料盘选择].行数-1;
			i行结束:=0;
			i列起始:=0;
			i列结束:=料盘配置[手动料盘选择].列数-1;
			i行递增:=-1;
			i列递增:=1;
		ELSIF ST_料盘配置V1_xg_0[手动料盘选择].x取料方位=3 THEN
			i行起始:=料盘配置[手动料盘选择].行数-1;
			i行结束:=0;
			i列起始:=料盘配置[手动料盘选择].列数-1;
			i列结束:=0;
			i行递增:=-1;
			i列递增:=-1;
		END_IF
		手动取料流程:=10;
END_IF

IF 手动取料流程=10 THEN

	FOR i:=i行起始 TO i行结束 BY i行递增 DO
		FOR j:=i列起始 TO i列结束 BY i列递增 DO
			IF 多料盘管理数据.料盘管理数据[手动料盘选择].屏蔽点位[i,j]=FALSE THEN
				IF 多料盘管理数据.料盘管理数据[手动料盘选择].点位状态[i,j]=E_点位状态.有料 THEN
					临时定位行号:=i;
					临时定位列号:=j;
					手动取料流程:=12;
					EXIT;
				END_IF

				IF i=i行结束 AND j=i列结束 THEN
					多料盘管理输出.错误:=TRUE;
					报错料盘:=手动料盘选择;
   					多料盘管理输出.错误信息 :=Standard.CONCAT(Standard.CONCAT('料盘', TO_STRING(手动料盘选择)), '没料了');
					多料盘管理输出.错误代码:=E_错误码.料盘取料空料;
				END_IF
			END_IF
		END_FOR

		IF 手动取料流程<>10 THEN
			EXIT;
		END_IF
	END_FOR

END_IF

IF 手动取料流程=12 THEN
	料盘轴运动输入.x定位位置:=料盘轴运动输入.目标位置[0]:=多料盘管理输出.目标X位置 := 料盘配置[手动料盘选择].起始X坐标 +
								临时定位列号 * 料盘配置[手动料盘选择].列间距 * x取料方向X +
								料盘配置[手动料盘选择].点位偏移[临时定位行号, 临时定位列号].x点位偏移;

	料盘轴运动输入.y定位位置:=料盘轴运动输入.目标位置[1]:=多料盘管理输出.目标Y位置 := 料盘配置[手动料盘选择].起始Y坐标 +
								临时定位行号 * 料盘配置[手动料盘选择].行间距 * x取料方向Y +
								料盘配置[手动料盘选择].点位偏移[临时定位行号, 临时定位列号].y点位偏移;

	料盘轴运动输入.z定位位置:=多料盘管理输出.目标Z位置 := 料盘配置[手动料盘选择].Z轴高度 +
								料盘配置[手动料盘选择].点位偏移[临时定位行号, 临时定位列号].z点位偏移;

// 	料盘轴运动输入.xy插补速度:=多料盘管理配置.xy插补速度;
// 	料盘轴运动输入.xy插补加速度:=多料盘管理配置.xy插补加速度;
// 	料盘轴运动输入.xy插补减速度:=多料盘管理配置.xy插补减速度;

	料盘轴运动输入.x定位速度:=多料盘管理配置.x速度;
	料盘轴运动输入.x定位加速度:=多料盘管理配置.x加速度;
	料盘轴运动输入.x定位减速度:=多料盘管理配置.x减速度;

	料盘轴运动输入.y定位速度:=多料盘管理配置.y速度;
	料盘轴运动输入.y定位加速度:=多料盘管理配置.y加速度;
	料盘轴运动输入.y定位减速度:=多料盘管理配置.y减速度;

	IF 料盘工艺配置[手动料盘选择].取料z轴下降减速动作.启用=1 THEN
		IF z轴.fActPosition>料盘工艺配置[手动料盘选择].取料z轴下降减速动作.取料减速位置 THEN
			料盘轴运动输入.z定位速度:= 料盘工艺配置[手动料盘选择].取料z轴下降减速动作.取料减速速度;
		ELSE
			料盘轴运动输入.z定位速度:=多料盘管理配置.z速度;
		END_IF
	ELSE
		料盘轴运动输入.z定位速度:=多料盘管理配置.z速度;
	END_IF

	料盘轴运动输入.z定位加速度:=多料盘管理配置.z加速度;
	料盘轴运动输入.z定位减速度:=多料盘管理配置.z减速度;

	IF x轴.nAxisState=Standstill  AND y轴.nAxisState=Standstill AND NOT 多料盘管理输入.暂停 THEN
		//料盘轴运动输入.插补启动:=TRUE;

		料盘轴运动输入.x轴定位:=TRUE;
		料盘轴运动输入.y轴定位:=TRUE;
		手动取料流程:=13;
	ELSIF 多料盘管理输入.暂停 THEN
		多料盘管理输出.暂停完成:=TRUE;
	END_IF
ELSIF 手动取料流程=13 THEN
	IF x轴.nAxisState=Standstill  AND y轴.nAxisState=Standstill AND NOT 多料盘管理输入.暂停 THEN
		//料盘轴运动输入.插补启动:=TRUE;

		料盘轴运动输入.x轴定位:=TRUE;
		料盘轴运动输入.y轴定位:=TRUE;
	//ELSIF 多料盘管理输入.暂停 THEN
	//	多料盘管理输出.暂停完成:=TRUE;
	END_IF
	IF 插补定位完成 AND x轴.nAxisState=Standstill  AND y轴.nAxisState=Standstill  THEN

		//料盘轴运动输入.插补启动:=FALSE;
		料盘轴运动输入.x轴定位:=FALSE;
		料盘轴运动输入.y轴定位:=FALSE;

		IF z轴.nAxisState=Standstill AND NOT 多料盘管理输入.暂停 THEN
			(* 移动轴 *)
			料盘轴运动输入.Z轴定位:=TRUE;
			手动取料流程:=14;
		ELSIF 多料盘管理输入.暂停 THEN
		多料盘管理输出.暂停完成:=TRUE;
		END_IF
	END_IF
END_IF

IF 手动取料流程=14 THEN
	IF z轴定位到位=FALSE AND z轴.nAxisState=Standstill AND NOT 多料盘管理输入.暂停 THEN
			(* 移动轴 *)
			料盘轴运动输入.Z轴定位:=TRUE;
			手动取料流程:=14;
	ELSIF z轴定位到位 AND 多料盘管理输入.暂停 THEN
		多料盘管理输出.暂停完成:=TRUE;
	END_IF
	IF 料盘工艺配置[手动料盘选择].取料z轴下降减速动作.启用=1 THEN
		IF z轴.fActPosition>料盘工艺配置[手动料盘选择].取料z轴下降减速动作.取料减速位置 THEN
			料盘轴运动输入.z定位速度:= 料盘工艺配置[手动料盘选择].取料z轴下降减速动作.取料减速速度;

		END_IF
	END_IF
	IF z轴定位到位 AND z轴.nAxisState=Standstill AND NOT 多料盘管理输入.暂停 THEN
		料盘轴运动输入.Z轴定位:=FALSE;

		IF 料盘工艺配置[手动料盘选择].取料附加动作.模式 =0 THEN
			多料盘管理数据.料盘管理数据[手动料盘选择].点位状态[临时定位行号,临时定位列号]:=E_点位状态.无料;
			多料盘管理输出.料盘运动状态:=E_料盘运动状态.待机;
			多料盘管理输出.到达定位位置:=TRUE;
			手动取料流程:=0;
		ELSIF 料盘工艺配置[手动料盘选择].取料附加动作.模式 =1 THEN
			手动取料流程:=20;
		END_IF
	END_IF
ELSIF 手动取料流程=20 THEN
	IF 料盘工艺配置[手动料盘选择].取料附加动作.索引=0 AND x轴.nAxisState=Standstill AND NOT 多料盘管理输入.暂停 THEN
		料盘轴运动输入.X定位位置:=多料盘管理输出.目标X位置 := 料盘工艺配置[手动料盘选择].取料附加动作.偏移值+x轴.fActPosition;
		料盘轴运动输入.x定位速度:= 料盘工艺配置[手动料盘选择].取料附加动作.速度;
		料盘轴运动输入.x定位加速度:= 料盘工艺配置[手动料盘选择].取料附加动作.加速度;
		料盘轴运动输入.x定位减速度:=料盘工艺配置[手动料盘选择].取料附加动作.减速度;
		料盘轴运动输入.x轴定位:=TRUE;
		手动取料流程:=30;
	ELSIF 料盘工艺配置[手动料盘选择].取料附加动作.索引=1 AND y轴.nAxisState=Standstill AND NOT 多料盘管理输入.暂停 THEN
		料盘轴运动输入.y定位位置:=多料盘管理输出.目标y位置 := 料盘工艺配置[手动料盘选择].取料附加动作.偏移值+y轴.fActPosition;
		料盘轴运动输入.y定位速度:=料盘工艺配置[手动料盘选择].取料附加动作.速度;
		料盘轴运动输入.y定位加速度:=料盘工艺配置[手动料盘选择].取料附加动作.加速度;
		料盘轴运动输入.y定位减速度:=料盘工艺配置[手动料盘选择].取料附加动作.减速度;
		料盘轴运动输入.y轴定位:=TRUE;
		手动取料流程:=30;
	ELSIF 料盘工艺配置[手动料盘选择].取料附加动作.索引=2 AND z轴.nAxisState=Standstill AND NOT 多料盘管理输入.暂停 THEN
		料盘轴运动输入.z定位位置:=多料盘管理输出.目标z位置 := 料盘工艺配置[手动料盘选择].取料附加动作.偏移值+z轴.fActPosition;
		料盘轴运动输入.z定位速度:=料盘工艺配置[手动料盘选择].取料附加动作.速度;
		料盘轴运动输入.z定位加速度:=料盘工艺配置[手动料盘选择].取料附加动作.加速度;
		料盘轴运动输入.z定位减速度:=料盘工艺配置[手动料盘选择].取料附加动作.减速度;
		料盘轴运动输入.z轴定位:=TRUE;
		手动取料流程:=30;
	ELSIF 多料盘管理输入.暂停 THEN
		多料盘管理输出.暂停完成:=TRUE;
	END_IF

ELSIF 手动取料流程=30 THEN
	IF 料盘工艺配置[手动料盘选择].取料附加动作.索引=0 THEN
		IF x轴定位到位 AND x轴.nAxisState=Standstill THEN
			多料盘管理数据.料盘管理数据[手动料盘选择].点位状态[临时定位行号,临时定位列号]:=E_点位状态.无料;
			料盘轴运动输入.x轴定位:=FALSE;
			多料盘管理输出.料盘运动状态:=E_料盘运动状态.待机;
			多料盘管理输出.到达定位位置:=TRUE;
			手动取料流程:=0;
		END_IF
	ELSIF 料盘工艺配置[手动料盘选择].取料附加动作.索引=1 THEN
		IF y轴定位到位 AND y轴.nAxisState=Standstill THEN
			多料盘管理数据.料盘管理数据[手动料盘选择].点位状态[临时定位行号,临时定位列号]:=E_点位状态.无料;
			料盘轴运动输入.y轴定位:=FALSE;
			多料盘管理输出.料盘运动状态:=E_料盘运动状态.待机;
			多料盘管理输出.到达定位位置:=TRUE;
			手动取料流程:=0;
		END_IF
	ELSIF 料盘工艺配置[手动料盘选择].取料附加动作.索引=2 THEN
		IF z轴定位到位 AND z轴.nAxisState=Standstill THEN
			多料盘管理数据.料盘管理数据[手动料盘选择].点位状态[临时定位行号,临时定位列号]:=E_点位状态.无料;
			料盘轴运动输入.z轴定位:=FALSE;
			多料盘管理输出.料盘运动状态:=E_料盘运动状态.待机;
			多料盘管理输出.到达定位位置:=TRUE;
			手动取料流程:=0;
		END_IF
	END_IF
END_IF

(* ---- FB_多料盘管理.ACT_手动指定取料.action.st ---- *)
手动指定取料上升沿(CLK:=S_多料盘管理输入HMI_xg_V1_0.指定取料 AND NOT 多料盘管理输入.手自动, Q=> );

IF 手动指定取料上升沿.Q AND 轴可运动 AND 流程可运行
THEN
	料盘轴运动输入.x轴定位:=FALSE;
	料盘轴运动输入.y轴定位:=FALSE;
	料盘轴运动输入.Z轴定位:=FALSE;
	料盘轴运动输入.插补启动:=FALSE;
	临时定位列号:=多料盘管理输入HMI.目标点位.列号;
	临时定位行号:=多料盘管理输入HMI.目标点位.行号;
	手动料盘选择:=多料盘管理输入hmi.料盘选择;
	指定取料流程:=2;
	多料盘管理输出.料盘运动状态:=E_料盘运动状态.指定取料中;

ELSE
	;
END_IF;

IF 指定取料流程=2 THEN
	IF z轴在待料位=FALSE THEN
		料盘轴运动输入.z定位位置:= 多料盘管理输出.目标Z位置 := 多料盘管理配置.z轴待料位;
		料盘轴运动输入.z定位速度:=多料盘管理配置.z速度;
		料盘轴运动输入.z定位加速度:=多料盘管理配置.z加速度;
		料盘轴运动输入.z定位减速度:=多料盘管理配置.z减速度;
		料盘轴运动输入.Z轴定位:=TRUE;
		指定取料流程:=5;
	ELSE
		指定取料流程:=5;
	END_IF
END_IF

IF 指定取料流程=5 THEN
	IF z轴在待料位=FALSE THEN
		料盘轴运动输入.z定位位置:= 多料盘管理输出.目标Z位置 := 多料盘管理配置.z轴待料位;
		料盘轴运动输入.z定位速度:=多料盘管理配置.z速度;
		料盘轴运动输入.z定位加速度:=多料盘管理配置.z加速度;
		料盘轴运动输入.z定位减速度:=多料盘管理配置.z减速度;
		料盘轴运动输入.Z轴定位:=TRUE;
	END_IF
	IF z轴在待料位 AND z轴.nAxisState=Standstill AND NOT 多料盘管理输入.暂停  THEN
		料盘轴运动输入.Z轴定位:=FALSE;
		指定取料流程:=6;
	ELSIF 多料盘管理输入.暂停 THEN
		多料盘管理输出.暂停完成:=TRUE;
	END_IF
END_IF

IF 指定取料流程=6 THEN
	IF FC_方向判断(
	i方向X:= x取料方向X,
	i方向Y:= x取料方向Y ,
	f起始点X:=料盘配置[手动料盘选择].起始X坐标 ,
	f起始点Y:= 料盘配置[手动料盘选择].起始Y坐标 ,
	f参考点X:=ST_料盘配置V1_xg_0[手动料盘选择].lf取料参考点x坐标 ,
	f参考点Y:=ST_料盘配置V1_xg_0[手动料盘选择].lf取料参考点y坐标 )=1 THEN
		多料盘管理输出.错误:=TRUE;
		报错料盘:=手动料盘选择;
		多料盘管理输出.错误信息 :=Standard.CONCAT(Standard.CONCAT('料盘', TO_STRING(手动料盘选择)), '取料参考点错误,不能和起始点相同');
		多料盘管理输出.错误代码:=E_错误码.取料参考点错误不能和起始点相同;
	ELSE
		指定取料流程:=12;
	END_IF
END_IF

IF 指定取料流程=12 THEN
	料盘轴运动输入.x定位位置:=料盘轴运动输入.目标位置[0]:=多料盘管理输出.目标X位置 := 料盘配置[手动料盘选择].起始X坐标 +
								临时定位列号 * 料盘配置[手动料盘选择].列间距 * x取料方向X +
								料盘配置[手动料盘选择].点位偏移[临时定位行号, 临时定位列号].x点位偏移;

	料盘轴运动输入.y定位位置:=料盘轴运动输入.目标位置[1]:=多料盘管理输出.目标Y位置 := 料盘配置[手动料盘选择].起始Y坐标 +
								临时定位行号 * 料盘配置[手动料盘选择].行间距 * x取料方向Y +
								料盘配置[手动料盘选择].点位偏移[临时定位行号, 临时定位列号].y点位偏移;

	料盘轴运动输入.z定位位置:=多料盘管理输出.目标Z位置 := 料盘配置[手动料盘选择].Z轴高度 +
								料盘配置[手动料盘选择].点位偏移[临时定位行号, 临时定位列号].z点位偏移;

// 	料盘轴运动输入.xy插补速度:=多料盘管理配置.xy插补速度;
// 	料盘轴运动输入.xy插补加速度:=多料盘管理配置.xy插补加速度;
// 	料盘轴运动输入.xy插补减速度:=多料盘管理配置.xy插补减速度;

	料盘轴运动输入.x定位速度:=多料盘管理配置.x速度;
	料盘轴运动输入.x定位加速度:=多料盘管理配置.x加速度;
	料盘轴运动输入.x定位减速度:=多料盘管理配置.x减速度;

	料盘轴运动输入.y定位速度:=多料盘管理配置.y速度;
	料盘轴运动输入.y定位加速度:=多料盘管理配置.y加速度;
	料盘轴运动输入.y定位减速度:=多料盘管理配置.y减速度;

	IF 料盘工艺配置[手动料盘选择].取料z轴下降减速动作.启用=1 THEN
		IF z轴.fActPosition>料盘工艺配置[手动料盘选择].取料z轴下降减速动作.取料减速位置 THEN
			料盘轴运动输入.z定位速度:= 料盘工艺配置[手动料盘选择].取料z轴下降减速动作.取料减速速度;
		ELSE
			料盘轴运动输入.z定位速度:=多料盘管理配置.z速度;
		END_IF
	ELSE
		料盘轴运动输入.z定位速度:=多料盘管理配置.z速度;
	END_IF

	料盘轴运动输入.z定位加速度:=多料盘管理配置.z加速度;
	料盘轴运动输入.z定位减速度:=多料盘管理配置.z减速度;

	IF x轴.nAxisState=Standstill  AND y轴.nAxisState=Standstill AND NOT 多料盘管理输入.暂停 THEN
		//料盘轴运动输入.插补启动:=TRUE;

		料盘轴运动输入.x轴定位:=TRUE;
		料盘轴运动输入.y轴定位:=TRUE;
		指定取料流程:=13;
	ELSIF 多料盘管理输入.暂停 THEN
		多料盘管理输出.暂停完成:=TRUE;
	END_IF
ELSIF 指定取料流程=13 THEN
	IF x轴.nAxisState=Standstill  AND y轴.nAxisState=Standstill AND NOT 多料盘管理输入.暂停 THEN
		//料盘轴运动输入.插补启动:=TRUE;

		料盘轴运动输入.x轴定位:=TRUE;
		料盘轴运动输入.y轴定位:=TRUE;
	//ELSIF 多料盘管理输入.暂停 THEN
	//	多料盘管理输出.暂停完成:=TRUE;
	END_IF
	IF 插补定位完成 AND x轴.nAxisState=Standstill  AND y轴.nAxisState=Standstill  THEN

		//料盘轴运动输入.插补启动:=FALSE;
		料盘轴运动输入.x轴定位:=FALSE;
		料盘轴运动输入.y轴定位:=FALSE;

		IF z轴.nAxisState=Standstill AND NOT 多料盘管理输入.暂停 THEN
			(* 移动轴 *)
			料盘轴运动输入.Z轴定位:=TRUE;
			指定取料流程:=14;
		ELSIF 多料盘管理输入.暂停 THEN
		多料盘管理输出.暂停完成:=TRUE;
		END_IF
	END_IF
END_IF

IF 指定取料流程=14 THEN
	IF z轴定位到位=FALSE AND z轴.nAxisState=Standstill AND NOT 多料盘管理输入.暂停 THEN
			(* 移动轴 *)
			料盘轴运动输入.Z轴定位:=TRUE;
			指定取料流程:=14;
	ELSIF z轴定位到位 AND 多料盘管理输入.暂停 THEN
		多料盘管理输出.暂停完成:=TRUE;
	END_IF
	IF 料盘工艺配置[手动料盘选择].取料z轴下降减速动作.启用=1 THEN
		IF z轴.fActPosition>料盘工艺配置[手动料盘选择].取料z轴下降减速动作.取料减速位置 THEN
			料盘轴运动输入.z定位速度:= 料盘工艺配置[手动料盘选择].取料z轴下降减速动作.取料减速速度;

		END_IF
	END_IF
	IF z轴定位到位 AND z轴.nAxisState=Standstill AND NOT 多料盘管理输入.暂停 THEN
		料盘轴运动输入.Z轴定位:=FALSE;

		IF 料盘工艺配置[手动料盘选择].取料附加动作.模式 =0 THEN
			多料盘管理数据.料盘管理数据[手动料盘选择].点位状态[临时定位行号,临时定位列号]:=E_点位状态.无料;
			多料盘管理输出.料盘运动状态:=E_料盘运动状态.待机;
			多料盘管理输出.到达定位位置:=TRUE;
			指定取料流程:=0;
		ELSIF 料盘工艺配置[手动料盘选择].取料附加动作.模式 =1 THEN
			指定取料流程:=20;
		END_IF
	END_IF
ELSIF 指定取料流程=20 THEN
	IF 料盘工艺配置[手动料盘选择].取料附加动作.索引=0 AND x轴.nAxisState=Standstill AND NOT 多料盘管理输入.暂停 THEN
		料盘轴运动输入.X定位位置:=多料盘管理输出.目标X位置 := 料盘工艺配置[手动料盘选择].取料附加动作.偏移值+x轴.fActPosition;
		料盘轴运动输入.x定位速度:= 料盘工艺配置[手动料盘选择].取料附加动作.速度;
		料盘轴运动输入.x定位加速度:= 料盘工艺配置[手动料盘选择].取料附加动作.加速度;
		料盘轴运动输入.x定位减速度:=料盘工艺配置[手动料盘选择].取料附加动作.减速度;
		料盘轴运动输入.x轴定位:=TRUE;
		指定取料流程:=30;
	ELSIF 料盘工艺配置[手动料盘选择].取料附加动作.索引=1 AND y轴.nAxisState=Standstill AND NOT 多料盘管理输入.暂停 THEN
		料盘轴运动输入.y定位位置:=多料盘管理输出.目标y位置 := 料盘工艺配置[手动料盘选择].取料附加动作.偏移值+y轴.fActPosition;
		料盘轴运动输入.y定位速度:=料盘工艺配置[手动料盘选择].取料附加动作.速度;
		料盘轴运动输入.y定位加速度:=料盘工艺配置[手动料盘选择].取料附加动作.加速度;
		料盘轴运动输入.y定位减速度:=料盘工艺配置[手动料盘选择].取料附加动作.减速度;
		料盘轴运动输入.y轴定位:=TRUE;
		指定取料流程:=30;
	ELSIF 料盘工艺配置[手动料盘选择].取料附加动作.索引=2 AND z轴.nAxisState=Standstill AND NOT 多料盘管理输入.暂停 THEN
		料盘轴运动输入.z定位位置:=多料盘管理输出.目标z位置 := 料盘工艺配置[手动料盘选择].取料附加动作.偏移值+z轴.fActPosition;
		料盘轴运动输入.z定位速度:=料盘工艺配置[手动料盘选择].取料附加动作.速度;
		料盘轴运动输入.z定位加速度:=料盘工艺配置[手动料盘选择].取料附加动作.加速度;
		料盘轴运动输入.z定位减速度:=料盘工艺配置[手动料盘选择].取料附加动作.减速度;
		料盘轴运动输入.z轴定位:=TRUE;
		指定取料流程:=30;
	ELSIF 多料盘管理输入.暂停 THEN
		多料盘管理输出.暂停完成:=TRUE;
	END_IF

ELSIF 指定取料流程=30 THEN
	IF 料盘工艺配置[手动料盘选择].取料附加动作.索引=0 THEN
		IF x轴定位到位 AND x轴.nAxisState=Standstill THEN
			多料盘管理数据.料盘管理数据[手动料盘选择].点位状态[临时定位行号,临时定位列号]:=E_点位状态.无料;
			料盘轴运动输入.x轴定位:=FALSE;
			多料盘管理输出.料盘运动状态:=E_料盘运动状态.待机;
			多料盘管理输出.到达定位位置:=TRUE;
			指定取料流程:=0;
		END_IF
	ELSIF 料盘工艺配置[手动料盘选择].取料附加动作.索引=1 THEN
		IF y轴定位到位 AND y轴.nAxisState=Standstill THEN
			多料盘管理数据.料盘管理数据[手动料盘选择].点位状态[临时定位行号,临时定位列号]:=E_点位状态.无料;
			料盘轴运动输入.y轴定位:=FALSE;
			多料盘管理输出.料盘运动状态:=E_料盘运动状态.待机;
			多料盘管理输出.到达定位位置:=TRUE;
			指定取料流程:=0;
		END_IF
	ELSIF 料盘工艺配置[手动料盘选择].取料附加动作.索引=2 THEN
		IF z轴定位到位 AND z轴.nAxisState=Standstill THEN
			多料盘管理数据.料盘管理数据[手动料盘选择].点位状态[临时定位行号,临时定位列号]:=E_点位状态.无料;
			料盘轴运动输入.z轴定位:=FALSE;
			多料盘管理输出.料盘运动状态:=E_料盘运动状态.待机;
			多料盘管理输出.到达定位位置:=TRUE;
			指定取料流程:=0;
		END_IF
	END_IF
END_IF

(* ---- FB_多料盘管理.ACT_手动指定放料.action.st ---- *)
手动指定放料上升沿(CLK:=S_多料盘管理输入HMI_xg_V1_0.指定放料 AND NOT 多料盘管理输入.手自动, Q=> );

IF 手动指定放料上升沿.Q AND 轴可运动 AND 流程可运行
THEN
	料盘轴运动输入.x轴定位:=FALSE;
	料盘轴运动输入.y轴定位:=FALSE;
	料盘轴运动输入.Z轴定位:=FALSE;
	料盘轴运动输入.插补启动:=FALSE;
	临时定位列号:=多料盘管理输入HMI.目标点位.列号;
	临时定位行号:=多料盘管理输入HMI.目标点位.行号;
	手动料盘选择:=多料盘管理输入hmi.料盘选择;
	指定放料流程:=2;
	多料盘管理输出.料盘运动状态:=E_料盘运动状态.指定放料中;

ELSE
	;
END_IF;

IF 指定放料流程=2 THEN
	IF z轴在待料位=FALSE THEN
		料盘轴运动输入.z定位位置:=多料盘管理输出.目标Z位置 := 多料盘管理配置.z轴待料位;
		料盘轴运动输入.z定位速度:=多料盘管理配置.z速度;
		料盘轴运动输入.z定位加速度:=多料盘管理配置.z加速度;
		料盘轴运动输入.z定位减速度:=多料盘管理配置.z减速度;
		料盘轴运动输入.Z轴定位:=TRUE;
		指定放料流程:=5;
	ELSE
		指定放料流程:=5;
	END_IF
END_IF

IF 指定放料流程=5 THEN
	IF z轴在待料位=FALSE THEN
		料盘轴运动输入.z定位位置:=多料盘管理输出.目标Z位置 := 多料盘管理配置.z轴待料位;
		料盘轴运动输入.z定位速度:=多料盘管理配置.z速度;
		料盘轴运动输入.z定位加速度:=多料盘管理配置.z加速度;
		料盘轴运动输入.z定位减速度:=多料盘管理配置.z减速度;
		料盘轴运动输入.Z轴定位:=TRUE;
	END_IF
	IF z轴在待料位 AND z轴.nAxisState=Standstill AND NOT 多料盘管理输入.暂停  THEN
		料盘轴运动输入.Z轴定位:=FALSE;
		指定放料流程:=6;
	ELSIF 多料盘管理输入.暂停 THEN
		多料盘管理输出.暂停完成:=TRUE;
	END_IF
END_IF

IF 指定放料流程=6 THEN
	IF FC_方向判断(
	i方向X:= x放料方向X,
	i方向Y:= x放料方向Y ,
	f起始点X:=料盘配置[手动料盘选择].放料起始X坐标 ,
	f起始点Y:= 料盘配置[手动料盘选择].放料起始Y坐标 ,
	f参考点X:=ST_料盘配置V1_xg_0[手动料盘选择].lf放料参考点x坐标 ,
	f参考点Y:=ST_料盘配置V1_xg_0[手动料盘选择].lf放料参考点y坐标 )=1 THEN
		多料盘管理输出.错误:=TRUE;
		报错料盘:=手动料盘选择;
		多料盘管理输出.错误信息 :=Standard.CONCAT(Standard.CONCAT('料盘', TO_STRING(手动料盘选择)), '放料参考点错误,不能和起始点相同');
		多料盘管理输出.错误代码:=E_错误码.放料参考点错误不能和起始点相同;
	ELSE
		指定放料流程:=12;
	END_IF
END_IF

IF 指定放料流程=12 THEN
	料盘轴运动输入.x定位位置:=料盘轴运动输入.目标位置[0]:=多料盘管理输出.目标X位置 := 料盘配置[手动料盘选择].放料起始X坐标 +
								临时定位列号 * 料盘配置[手动料盘选择].列间距 *x放料方向X +
								料盘配置[手动料盘选择].点位偏移[临时定位行号, 临时定位列号].x点位偏移;

	料盘轴运动输入.y定位位置:=料盘轴运动输入.目标位置[1]:=多料盘管理输出.目标Y位置 := 料盘配置[手动料盘选择].放料起始Y坐标 +
								临时定位行号 * 料盘配置[手动料盘选择].行间距 *x放料方向Y +
								料盘配置[手动料盘选择].点位偏移[临时定位行号, 临时定位列号].y点位偏移;

	料盘轴运动输入.z定位位置:=多料盘管理输出.目标Z位置 := 料盘配置[手动料盘选择].放料Z轴高度 +
								料盘配置[手动料盘选择].点位偏移[临时定位行号, 临时定位列号].z点位偏移;

// 	料盘轴运动输入.xy插补速度:=多料盘管理配置.xy插补速度;
// 	料盘轴运动输入.xy插补加速度:=多料盘管理配置.xy插补加速度;
// 	料盘轴运动输入.xy插补减速度:=多料盘管理配置.xy插补减速度;

	料盘轴运动输入.x定位速度:=多料盘管理配置.x速度;
	料盘轴运动输入.x定位加速度:=多料盘管理配置.x加速度;
	料盘轴运动输入.x定位减速度:=多料盘管理配置.x减速度;

	料盘轴运动输入.y定位速度:=多料盘管理配置.y速度;
	料盘轴运动输入.y定位加速度:=多料盘管理配置.y加速度;
	料盘轴运动输入.y定位减速度:=多料盘管理配置.y减速度;

	IF 料盘工艺配置[手动料盘选择].放料z轴下降减速动作.启用=1 THEN
		IF z轴.fActPosition>料盘工艺配置[手动料盘选择].放料z轴下降减速动作.放料减速位置 THEN
			料盘轴运动输入.z定位速度:= 料盘工艺配置[手动料盘选择].放料z轴下降减速动作.放料减速速度;
		ELSE
			料盘轴运动输入.z定位速度:=多料盘管理配置.z速度;
		END_IF
	ELSE
		料盘轴运动输入.z定位速度:=多料盘管理配置.z速度;
	END_IF
	料盘轴运动输入.z定位加速度:=多料盘管理配置.z加速度;
	料盘轴运动输入.z定位减速度:=多料盘管理配置.z减速度;

	IF x轴.nAxisState=Standstill  AND y轴.nAxisState=Standstill AND NOT 多料盘管理输入.暂停 THEN
		//料盘轴运动输入.插补启动:=TRUE;
		料盘轴运动输入.x轴定位:=TRUE;
		料盘轴运动输入.y轴定位:=TRUE;
		指定放料流程:=13;
	ELSIF 多料盘管理输入.暂停 THEN
		多料盘管理输出.暂停完成:=TRUE;
	END_IF

ELSIF 指定放料流程=13 THEN
	IF x轴.nAxisState=Standstill  AND y轴.nAxisState=Standstill AND NOT 多料盘管理输入.暂停 THEN
		//料盘轴运动输入.插补启动:=TRUE;
		料盘轴运动输入.x轴定位:=TRUE;
		料盘轴运动输入.y轴定位:=TRUE;
	//ELSIF 多料盘管理输入.暂停 THEN
	//	多料盘管理输出.暂停完成:=TRUE;
	END_IF
	IF 插补定位完成 AND x轴.nAxisState=Standstill  AND y轴.nAxisState=Standstill  THEN

		//料盘轴运动输入.插补启动:=FALSE;
		料盘轴运动输入.x轴定位:=FALSE;
		料盘轴运动输入.y轴定位:=FALSE;

		IF z轴.nAxisState=Standstill AND NOT 多料盘管理输入.暂停  THEN
			料盘轴运动输入.Z轴定位:=TRUE;
			指定放料流程:=14;
		ELSIF 多料盘管理输入.暂停 THEN
			多料盘管理输出.暂停完成:=TRUE;
		END_IF
	END_IF
END_IF

IF 指定放料流程=14 THEN
	IF z轴定位到位=FALSE AND z轴.nAxisState=Standstill AND NOT 多料盘管理输入.暂停  THEN
			料盘轴运动输入.Z轴定位:=TRUE;
		ELSIF z轴定位到位 AND 多料盘管理输入.暂停 THEN
			多料盘管理输出.暂停完成:=TRUE;
		END_IF
	IF 料盘工艺配置[手动料盘选择].放料z轴下降减速动作.启用=1 THEN
		IF z轴.fActPosition>料盘工艺配置[手动料盘选择].放料z轴下降减速动作.放料减速位置 THEN
			料盘轴运动输入.z定位速度:= 料盘工艺配置[手动料盘选择].放料z轴下降减速动作.放料减速速度;

		END_IF

	END_IF

	IF z轴定位到位 AND z轴.nAxisState=Standstill AND NOT 多料盘管理输入.暂停  THEN
		料盘轴运动输入.Z轴定位:=FALSE;

		IF 料盘工艺配置[手动料盘选择].放料附加动作.模式 =0 THEN
			多料盘管理数据.料盘管理数据[手动料盘选择].点位状态[临时定位行号,临时定位列号]:=E_点位状态.有料;
			多料盘管理输出.料盘运动状态:=E_料盘运动状态.待机;
			多料盘管理输出.到达定位位置:=TRUE;
			指定放料流程:=0;
		ELSIF 料盘工艺配置[手动料盘选择].放料附加动作.模式 =1 THEN
			指定放料流程:=20;
		END_IF
	END_IF
ELSIF 指定放料流程=20 THEN
	IF 料盘工艺配置[手动料盘选择].放料附加动作.索引=0 AND x轴.nAxisState=Standstill AND NOT 多料盘管理输入.暂停 THEN
		料盘轴运动输入.X定位位置:=多料盘管理输出.目标X位置 := 料盘工艺配置[手动料盘选择].放料附加动作.偏移值+x轴.fActPosition;
		料盘轴运动输入.x定位速度:= 料盘工艺配置[手动料盘选择].放料附加动作.速度;
		料盘轴运动输入.x定位加速度:= 料盘工艺配置[手动料盘选择].放料附加动作.加速度;
		料盘轴运动输入.x定位减速度:=料盘工艺配置[手动料盘选择].放料附加动作.减速度;
		料盘轴运动输入.x轴定位:=TRUE;
		指定放料流程:=30;
	ELSIF 料盘工艺配置[手动料盘选择].放料附加动作.索引=1 AND y轴.nAxisState=Standstill AND NOT 多料盘管理输入.暂停  THEN
		料盘轴运动输入.y定位位置:=多料盘管理输出.目标y位置 := 料盘工艺配置[手动料盘选择].放料附加动作.偏移值+y轴.fActPosition;
		料盘轴运动输入.y定位速度:=料盘工艺配置[手动料盘选择].放料附加动作.速度;
		料盘轴运动输入.y定位加速度:=料盘工艺配置[手动料盘选择].放料附加动作.加速度;
		料盘轴运动输入.y定位减速度:=料盘工艺配置[手动料盘选择].放料附加动作.减速度;
		料盘轴运动输入.y轴定位:=TRUE;
		指定放料流程:=30;
	ELSIF 料盘工艺配置[手动料盘选择].放料附加动作.索引=2 AND z轴.nAxisState=Standstill AND NOT 多料盘管理输入.暂停  THEN
		料盘轴运动输入.z定位位置:=多料盘管理输出.目标z位置 := 料盘工艺配置[手动料盘选择].放料附加动作.偏移值+z轴.fActPosition;
		料盘轴运动输入.z定位速度:=料盘工艺配置[手动料盘选择].放料附加动作.速度;
		料盘轴运动输入.z定位加速度:=料盘工艺配置[手动料盘选择].放料附加动作.加速度;
		料盘轴运动输入.z定位减速度:=料盘工艺配置[手动料盘选择].放料附加动作.减速度;
		料盘轴运动输入.z轴定位:=TRUE;
		指定放料流程:=30;
	ELSIF 多料盘管理输入.暂停 THEN
		多料盘管理输出.暂停完成:=TRUE;
	END_IF

ELSIF 指定放料流程=30 THEN
	IF 料盘工艺配置[手动料盘选择].放料附加动作.索引=0 THEN
		IF x轴定位到位 AND x轴.nAxisState=Standstill THEN
			多料盘管理数据.料盘管理数据[手动料盘选择].点位状态[临时定位行号,临时定位列号]:=E_点位状态.有料;
			料盘轴运动输入.x轴定位:=FALSE;
			多料盘管理输出.料盘运动状态:=E_料盘运动状态.待机;
			多料盘管理输出.到达定位位置:=TRUE;
			指定放料流程:=0;
		END_IF
	ELSIF 料盘工艺配置[手动料盘选择].放料附加动作.索引=1 THEN
		IF y轴定位到位 AND y轴.nAxisState=Standstill  THEN
			多料盘管理数据.料盘管理数据[手动料盘选择].点位状态[临时定位行号,临时定位列号]:=E_点位状态.有料;
			料盘轴运动输入.y轴定位:=FALSE;
			多料盘管理输出.料盘运动状态:=E_料盘运动状态.待机;
			多料盘管理输出.到达定位位置:=TRUE;
			指定放料流程:=0;
		END_IF
	ELSIF 料盘工艺配置[手动料盘选择].放料附加动作.索引=2 THEN
		IF z轴定位到位 AND z轴.nAxisState=Standstill THEN
			多料盘管理数据.料盘管理数据[手动料盘选择].点位状态[临时定位行号,临时定位列号]:=E_点位状态.有料;
			料盘轴运动输入.z轴定位:=FALSE;
			多料盘管理输出.料盘运动状态:=E_料盘运动状态.待机;
			多料盘管理输出.到达定位位置:=TRUE;
			指定放料流程:=0;
		END_IF
	END_IF
END_IF

(* ---- FB_多料盘管理.ACT_手动放料.action.st ---- *)
手动放料上升沿(CLK:=S_多料盘管理输入HMI_xg_V1_0.放料 AND NOT 多料盘管理输入.手自动, Q=> );

IF 手动放料上升沿.Q AND 轴可运动 AND 流程可运行
THEN
	料盘轴运动输入.x轴定位:=FALSE;
	料盘轴运动输入.y轴定位:=FALSE;
	料盘轴运动输入.Z轴定位:=FALSE;
	料盘轴运动输入.插补启动:=FALSE;
	手动料盘选择:=多料盘管理输入hmi.料盘选择;;
	手动放料流程:=2;
	多料盘管理输出.料盘运动状态:=E_料盘运动状态.手动放料中;

ELSE
	;
END_IF;

IF 手动放料流程=2 THEN
	IF z轴在待料位=FALSE THEN
		料盘轴运动输入.z定位位置:=多料盘管理输出.目标Z位置 := 多料盘管理配置.z轴待料位;
		料盘轴运动输入.z定位速度:=多料盘管理配置.z速度;
		料盘轴运动输入.z定位加速度:=多料盘管理配置.z加速度;
		料盘轴运动输入.z定位减速度:=多料盘管理配置.z减速度;
		料盘轴运动输入.Z轴定位:=TRUE;
		手动放料流程:=5;
	ELSE
		手动放料流程:=5;
	END_IF
END_IF

IF 手动放料流程=5 THEN
	IF z轴在待料位=FALSE THEN
		料盘轴运动输入.z定位位置:=多料盘管理输出.目标Z位置 := 多料盘管理配置.z轴待料位;
		料盘轴运动输入.z定位速度:=多料盘管理配置.z速度;
		料盘轴运动输入.z定位加速度:=多料盘管理配置.z加速度;
		料盘轴运动输入.z定位减速度:=多料盘管理配置.z减速度;
		料盘轴运动输入.Z轴定位:=TRUE;
	END_IF
	IF z轴在待料位 AND z轴.nAxisState=Standstill AND NOT 多料盘管理输入.暂停  THEN
		料盘轴运动输入.Z轴定位:=FALSE;
		手动放料流程:=6;
	ELSIF 多料盘管理输入.暂停 THEN
		多料盘管理输出.暂停完成:=TRUE;
	END_IF
END_IF

IF 手动放料流程=6 THEN
	IF FC_方向判断(
	i方向X:= x放料方向X,
	i方向Y:= x放料方向Y ,
	f起始点X:=料盘配置[手动料盘选择].放料起始X坐标 ,
	f起始点Y:= 料盘配置[手动料盘选择].放料起始Y坐标 ,
	f参考点X:=ST_料盘配置V1_xg_0[手动料盘选择].lf放料参考点x坐标 ,
	f参考点Y:=ST_料盘配置V1_xg_0[手动料盘选择].lf放料参考点y坐标 )=1 THEN
		多料盘管理输出.错误:=TRUE;
		报错料盘:=手动料盘选择;
		多料盘管理输出.错误信息 :=Standard.CONCAT(Standard.CONCAT('料盘', TO_STRING(手动料盘选择)), '放料参考点错误,不能和起始点相同');
		多料盘管理输出.错误代码:=E_错误码.放料参考点错误不能和起始点相同;
	ELSE
		手动放料流程:=7;
	END_IF
END_IF

IF 手动放料流程=7 THEN
	//左上
		IF ST_料盘配置V1_xg_0[手动料盘选择].x放料方位=0 THEN
			i行起始:=0;
			i行结束:=料盘配置[手动料盘选择].行数-1;
			i列起始:=0;
			i列结束:=料盘配置[手动料盘选择].列数-1;
			i行递增:=1;
			i列递增:=1;
		ELSIF ST_料盘配置V1_xg_0[手动料盘选择].x放料方位=1 THEN
			i行起始:=0;
			i行结束:=料盘配置[手动料盘选择].行数-1;
			i列起始:=料盘配置[手动料盘选择].列数-1;
			i列结束:=0;
			i行递增:=1;
			i列递增:=-1;
		ELSIF ST_料盘配置V1_xg_0[手动料盘选择].x放料方位=2 THEN
			i行起始:=料盘配置[手动料盘选择].行数-1;
			i行结束:=0;
			i列起始:=0;
			i列结束:=料盘配置[手动料盘选择].列数-1;
			i行递增:=-1;
			i列递增:=1;
		ELSIF ST_料盘配置V1_xg_0[手动料盘选择].x放料方位=3 THEN
			i行起始:=料盘配置[手动料盘选择].行数-1;
			i行结束:=0;
			i列起始:=料盘配置[手动料盘选择].列数-1;
			i列结束:=0;
			i行递增:=-1;
			i列递增:=-1;
		END_IF
		手动放料流程:=10;
END_IF

IF 手动放料流程=10 THEN

	FOR i:=i行起始 TO i行结束 BY i行递增 DO
		FOR j:=i列起始 TO i列结束 BY i列递增 DO
			IF 多料盘管理数据.料盘管理数据[手动料盘选择].屏蔽点位[i,j]=FALSE THEN

				IF 多料盘管理数据.料盘管理数据[手动料盘选择].点位状态[i,j]=E_点位状态.无料 THEN
					临时定位行号:=i;
					临时定位列号:=j;
					手动放料流程:=12;
					EXIT;
				END_IF

				IF i=i行结束 AND j=i列结束 THEN
					多料盘管理输出.错误:=TRUE;
					报错料盘:=手动料盘选择;
   					多料盘管理输出.错误信息 :=Standard.CONCAT(Standard.CONCAT('料盘', TO_STRING(手动料盘选择)), '料满了');
					多料盘管理输出.错误代码:=E_错误码.料盘放料满料;
				END_IF
			END_IF
		END_FOR

		IF 手动放料流程<>10 THEN
			EXIT;
		END_IF
	END_FOR
END_IF

IF 手动放料流程=12 THEN
	料盘轴运动输入.x定位位置:=料盘轴运动输入.目标位置[0]:=多料盘管理输出.目标X位置 := 料盘配置[手动料盘选择].放料起始X坐标 +
								临时定位列号 * 料盘配置[手动料盘选择].列间距 *x放料方向X +
								料盘配置[手动料盘选择].点位偏移[临时定位行号, 临时定位列号].x点位偏移;

	料盘轴运动输入.y定位位置:=料盘轴运动输入.目标位置[1]:=多料盘管理输出.目标Y位置 := 料盘配置[手动料盘选择].放料起始Y坐标 +
								临时定位行号 * 料盘配置[手动料盘选择].行间距 *x放料方向Y +
								料盘配置[手动料盘选择].点位偏移[临时定位行号, 临时定位列号].y点位偏移;

	料盘轴运动输入.z定位位置:=多料盘管理输出.目标Z位置 := 料盘配置[手动料盘选择].放料Z轴高度 +
								料盘配置[手动料盘选择].点位偏移[临时定位行号, 临时定位列号].z点位偏移;

// 	料盘轴运动输入.xy插补速度:=多料盘管理配置.xy插补速度;
// 	料盘轴运动输入.xy插补加速度:=多料盘管理配置.xy插补加速度;
// 	料盘轴运动输入.xy插补减速度:=多料盘管理配置.xy插补减速度;

	料盘轴运动输入.x定位速度:=多料盘管理配置.x速度;
	料盘轴运动输入.x定位加速度:=多料盘管理配置.x加速度;
	料盘轴运动输入.x定位减速度:=多料盘管理配置.x减速度;

	料盘轴运动输入.y定位速度:=多料盘管理配置.y速度;
	料盘轴运动输入.y定位加速度:=多料盘管理配置.y加速度;
	料盘轴运动输入.y定位减速度:=多料盘管理配置.y减速度;

	IF 料盘工艺配置[手动料盘选择].放料z轴下降减速动作.启用=1 THEN
		IF z轴.fActPosition>料盘工艺配置[手动料盘选择].放料z轴下降减速动作.放料减速位置 THEN
			料盘轴运动输入.z定位速度:= 料盘工艺配置[手动料盘选择].放料z轴下降减速动作.放料减速速度;
		ELSE
			料盘轴运动输入.z定位速度:=多料盘管理配置.z速度;
		END_IF
	ELSE
		料盘轴运动输入.z定位速度:=多料盘管理配置.z速度;
	END_IF
	料盘轴运动输入.z定位加速度:=多料盘管理配置.z加速度;
	料盘轴运动输入.z定位减速度:=多料盘管理配置.z减速度;

	IF x轴.nAxisState=Standstill  AND y轴.nAxisState=Standstill AND NOT 多料盘管理输入.暂停 THEN
		//料盘轴运动输入.插补启动:=TRUE;
		料盘轴运动输入.x轴定位:=TRUE;
		料盘轴运动输入.y轴定位:=TRUE;
		手动放料流程:=13;
	ELSIF 多料盘管理输入.暂停 THEN
		多料盘管理输出.暂停完成:=TRUE;
	END_IF

ELSIF 手动放料流程=13 THEN
	IF x轴.nAxisState=Standstill  AND y轴.nAxisState=Standstill AND NOT 多料盘管理输入.暂停 THEN
		//料盘轴运动输入.插补启动:=TRUE;
		料盘轴运动输入.x轴定位:=TRUE;
		料盘轴运动输入.y轴定位:=TRUE;
	//ELSIF 多料盘管理输入.暂停 THEN
	//	多料盘管理输出.暂停完成:=TRUE;
	END_IF
	IF 插补定位完成 AND x轴.nAxisState=Standstill  AND y轴.nAxisState=Standstill  THEN

		//料盘轴运动输入.插补启动:=FALSE;
		料盘轴运动输入.x轴定位:=FALSE;
		料盘轴运动输入.y轴定位:=FALSE;

		IF z轴.nAxisState=Standstill AND NOT 多料盘管理输入.暂停  THEN
			料盘轴运动输入.Z轴定位:=TRUE;
			手动放料流程:=14;
		ELSIF 多料盘管理输入.暂停 THEN
			多料盘管理输出.暂停完成:=TRUE;
		END_IF
	END_IF
END_IF

IF 手动放料流程=14 THEN
	IF z轴定位到位=FALSE AND z轴.nAxisState=Standstill AND NOT 多料盘管理输入.暂停  THEN
			料盘轴运动输入.Z轴定位:=TRUE;
		ELSIF z轴定位到位 AND 多料盘管理输入.暂停 THEN
			多料盘管理输出.暂停完成:=TRUE;
		END_IF
	IF 料盘工艺配置[手动料盘选择].放料z轴下降减速动作.启用=1 THEN
		IF z轴.fActPosition>料盘工艺配置[手动料盘选择].放料z轴下降减速动作.放料减速位置 THEN
			料盘轴运动输入.z定位速度:= 料盘工艺配置[手动料盘选择].放料z轴下降减速动作.放料减速速度;

		END_IF

	END_IF

	IF z轴定位到位 AND z轴.nAxisState=Standstill AND NOT 多料盘管理输入.暂停  THEN
		料盘轴运动输入.Z轴定位:=FALSE;

		IF 料盘工艺配置[手动料盘选择].放料附加动作.模式 =0 THEN
			多料盘管理数据.料盘管理数据[手动料盘选择].点位状态[临时定位行号,临时定位列号]:=E_点位状态.有料;
			多料盘管理输出.料盘运动状态:=E_料盘运动状态.待机;
			多料盘管理输出.到达定位位置:=TRUE;
			手动放料流程:=0;
		ELSIF 料盘工艺配置[手动料盘选择].放料附加动作.模式 =1 THEN
			手动放料流程:=20;
		END_IF
	END_IF
ELSIF 手动放料流程=20 THEN
	IF 料盘工艺配置[手动料盘选择].放料附加动作.索引=0 AND x轴.nAxisState=Standstill AND NOT 多料盘管理输入.暂停 THEN
		料盘轴运动输入.X定位位置:=多料盘管理输出.目标X位置 := 料盘工艺配置[手动料盘选择].放料附加动作.偏移值+x轴.fActPosition;
		料盘轴运动输入.x定位速度:= 料盘工艺配置[手动料盘选择].放料附加动作.速度;
		料盘轴运动输入.x定位加速度:= 料盘工艺配置[手动料盘选择].放料附加动作.加速度;
		料盘轴运动输入.x定位减速度:=料盘工艺配置[手动料盘选择].放料附加动作.减速度;
		料盘轴运动输入.x轴定位:=TRUE;
		手动放料流程:=30;
	ELSIF 料盘工艺配置[手动料盘选择].放料附加动作.索引=1 AND y轴.nAxisState=Standstill AND NOT 多料盘管理输入.暂停  THEN
		料盘轴运动输入.y定位位置:=多料盘管理输出.目标y位置 := 料盘工艺配置[手动料盘选择].放料附加动作.偏移值+y轴.fActPosition;
		料盘轴运动输入.y定位速度:=料盘工艺配置[手动料盘选择].放料附加动作.速度;
		料盘轴运动输入.y定位加速度:=料盘工艺配置[手动料盘选择].放料附加动作.加速度;
		料盘轴运动输入.y定位减速度:=料盘工艺配置[手动料盘选择].放料附加动作.减速度;
		料盘轴运动输入.y轴定位:=TRUE;
		手动放料流程:=30;
	ELSIF 料盘工艺配置[手动料盘选择].放料附加动作.索引=2 AND z轴.nAxisState=Standstill AND NOT 多料盘管理输入.暂停  THEN
		料盘轴运动输入.z定位位置:=多料盘管理输出.目标z位置 := 料盘工艺配置[手动料盘选择].放料附加动作.偏移值+z轴.fActPosition;
		料盘轴运动输入.z定位速度:=料盘工艺配置[手动料盘选择].放料附加动作.速度;
		料盘轴运动输入.z定位加速度:=料盘工艺配置[手动料盘选择].放料附加动作.加速度;
		料盘轴运动输入.z定位减速度:=料盘工艺配置[手动料盘选择].放料附加动作.减速度;
		料盘轴运动输入.z轴定位:=TRUE;
		手动放料流程:=30;
	ELSIF 多料盘管理输入.暂停 THEN
		多料盘管理输出.暂停完成:=TRUE;
	END_IF

ELSIF 手动放料流程=30 THEN
	IF 料盘工艺配置[手动料盘选择].放料附加动作.索引=0 THEN
		IF x轴定位到位 AND x轴.nAxisState=Standstill THEN
			多料盘管理数据.料盘管理数据[手动料盘选择].点位状态[临时定位行号,临时定位列号]:=E_点位状态.有料;
			料盘轴运动输入.x轴定位:=FALSE;
			多料盘管理输出.料盘运动状态:=E_料盘运动状态.待机;
			多料盘管理输出.到达定位位置:=TRUE;
			手动放料流程:=0;
		END_IF
	ELSIF 料盘工艺配置[手动料盘选择].放料附加动作.索引=1 THEN
		IF y轴定位到位 AND y轴.nAxisState=Standstill  THEN
			多料盘管理数据.料盘管理数据[手动料盘选择].点位状态[临时定位行号,临时定位列号]:=E_点位状态.有料;
			料盘轴运动输入.y轴定位:=FALSE;
			多料盘管理输出.料盘运动状态:=E_料盘运动状态.待机;
			多料盘管理输出.到达定位位置:=TRUE;
			手动放料流程:=0;
		END_IF
	ELSIF 料盘工艺配置[手动料盘选择].放料附加动作.索引=2 THEN
		IF z轴定位到位 AND z轴.nAxisState=Standstill THEN
			多料盘管理数据.料盘管理数据[手动料盘选择].点位状态[临时定位行号,临时定位列号]:=E_点位状态.有料;
			料盘轴运动输入.z轴定位:=FALSE;
			多料盘管理输出.料盘运动状态:=E_料盘运动状态.待机;
			多料盘管理输出.到达定位位置:=TRUE;
			手动放料流程:=0;
		END_IF
	END_IF
END_IF

(* ---- FB_多料盘管理.ACT_料盘状态.action.st ---- *)
(* 更新料盘状态输出 *)
    FOR i := 0 TO GVL_常量.最大料盘数量 - 1 DO
        (* 检查料盘是否满料 *)
        多料盘管理输出.料盘管理输出[i].满料信号 := TRUE;  // 初始设为满料
        FOR row := 0 TO 料盘配置[i].行数 - 1 DO
            FOR col := 0 TO 料盘配置[i].列数 - 1 DO
                IF 多料盘管理数据.料盘管理数据[i].点位状态[row, col] = E_点位状态.无料 AND
                   NOT 多料盘管理数据.料盘管理数据[i].屏蔽点位[row, col] THEN
                    多料盘管理输出.料盘管理输出[i].满料信号 := FALSE;
                END_IF;
            END_FOR;
        END_FOR;

        (* 检查料盘是否无料 *)
        多料盘管理输出.料盘管理输出[i].无料信号 := TRUE;  // 初始设为无料
        FOR row := 0 TO 料盘配置[i].行数 - 1 DO
            FOR col := 0 TO 料盘配置[i].列数 - 1 DO
                IF 多料盘管理数据.料盘管理数据[i].点位状态[row, col] = E_点位状态.有料 AND
                   NOT 多料盘管理数据.料盘管理数据[i].屏蔽点位[row, col] THEN
                    多料盘管理输出.料盘管理输出[i].无料信号 := FALSE;
                END_IF;
            END_FOR;
        END_FOR;

        (* 输出当前点位坐标 *)
        多料盘管理输出.料盘管理输出[i].当前点位坐标.行号 := 临时定位行号;
		多料盘管理输出.料盘管理输出[i].当前点位坐标.列号 := 临时定位列号;
    END_FOR;

多料盘管理输出.当前X位置:=TO_REAL(x轴.fActPosition);
多料盘管理输出.当前y位置:=TO_REAL(y轴.fActPosition);
多料盘管理输出.当前z位置:=TO_REAL(z轴.fActPosition);

多料盘管理输出.当前X速度:=TO_REAL(x轴.fActVelocity);
多料盘管理输出.当前y速度:=TO_REAL(y轴.fActVelocity);
多料盘管理输出.当前z速度:=TO_REAL(z轴.fActVelocity);

(* ---- FB_多料盘管理.ACT_自动取料.action.st ---- *)
取料上升沿(CLK:=多料盘管理输入.取料 AND 多料盘管理输入.手自动, Q=> );
取料完成上升沿(CLK:=多料盘管理输入.取料完成 AND 多料盘管理输入.手自动, Q=> );

IF GVL_系统变量.全局状态=E_系统运行状态.系统状态_故障 THEN
	料盘轴运动输入.x轴定位:=FALSE;
	料盘轴运动输入.y轴定位:=FALSE;
	料盘轴运动输入.Z轴定位:=FALSE;
	料盘轴运动输入.插补启动:=FALSE;
	RETURN;
END_IF

IF GVL_系统变量.全局状态<>E_系统运行状态.系统状态_运行 AND GVL_系统变量.全局状态<>E_系统运行状态.系统状态_清料中  AND GVL_系统变量.全局状态<>E_系统运行状态.系统状态_暂停中 THEN

	RETURN;
END_IF

IF 取料完成上升沿.q THEN
	多料盘管理数据.料盘管理数据[多料盘管理输入.料盘选择].点位状态[临时定位行号,临时定位列号]:=E_点位状态.无料;
END_IF

IF 取料上升沿.Q AND 轴可运动 AND 流程可运行
	AND NOT 多料盘管理输入.到初始位 AND NOT 多料盘管理输入.放料 AND NOT 多料盘管理输入.定位
	 AND NOT 多料盘管理输入.暂停 AND NOT 多料盘管理输出.错误 AND
	(多料盘管理输出.料盘运动状态=E_料盘运动状态.待机
	OR 多料盘管理输出.料盘运动状态=E_料盘运动状态.暂停)
THEN
	料盘轴运动输入.x轴定位:=FALSE;
	料盘轴运动输入.y轴定位:=FALSE;
	料盘轴运动输入.Z轴定位:=FALSE;
	料盘轴运动输入.插补启动:=FALSE;
	多料盘管理输出.到达定位位置:=FALSE;
	IF 多料盘管理输出.料盘运动状态=E_料盘运动状态.暂停 THEN
		多料盘管理输出.料盘运动状态:=E_料盘运动状态.到取料位中;
		取料流程:=12;
	ELSE
		多料盘管理输出.料盘运动状态:=E_料盘运动状态.到取料位中;
		取料流程:=2;
	END_IF

ELSE
	;
END_IF;

IF 取料流程=2 THEN
	IF z轴在待料位=FALSE THEN
		料盘轴运动输入.z定位位置:= 多料盘管理输出.目标Z位置 := 多料盘管理配置.z轴待料位;
		料盘轴运动输入.z定位速度:=多料盘管理配置.z速度;
		料盘轴运动输入.z定位加速度:=多料盘管理配置.z加速度;
		料盘轴运动输入.z定位减速度:=多料盘管理配置.z减速度;
		料盘轴运动输入.Z轴定位:=TRUE;
		取料流程:=5;
	ELSE
		取料流程:=5;
	END_IF
END_IF

IF 取料流程=5 THEN
	IF z轴在待料位=FALSE AND NOT 多料盘管理输入.暂停 THEN
		料盘轴运动输入.z定位位置:= 多料盘管理输出.目标Z位置 := 多料盘管理配置.z轴待料位;
		料盘轴运动输入.z定位速度:=多料盘管理配置.z速度;
		料盘轴运动输入.z定位加速度:=多料盘管理配置.z加速度;
		料盘轴运动输入.z定位减速度:=多料盘管理配置.z减速度;
		料盘轴运动输入.Z轴定位:=TRUE;
	END_IF
	IF z轴在待料位 AND z轴.nAxisState=Standstill AND NOT 多料盘管理输入.暂停  THEN
		料盘轴运动输入.Z轴定位:=FALSE;
		取料流程:=6;
	ELSIF 多料盘管理输入.暂停 THEN
		多料盘管理输出.暂停完成:=TRUE;
	END_IF
END_IF

IF 取料流程=6 THEN
	IF FC_方向判断(
	i方向X:= x取料方向X,
	i方向Y:= x取料方向Y ,
	f起始点X:=料盘配置[多料盘管理输入.料盘选择].起始X坐标 ,
	f起始点Y:= 料盘配置[多料盘管理输入.料盘选择].起始Y坐标 ,
	f参考点X:=ST_料盘配置V1_xg_0[多料盘管理输入.料盘选择].lf取料参考点x坐标 ,
	f参考点Y:=ST_料盘配置V1_xg_0[多料盘管理输入.料盘选择].lf取料参考点y坐标 )=1 THEN
		多料盘管理输出.错误:=TRUE;
		报错料盘:=多料盘管理输入.料盘选择;
		多料盘管理输出.错误信息 :=Standard.CONCAT(Standard.CONCAT('料盘', TO_STRING(多料盘管理输入.料盘选择)), '取料参考点错误,不能和起始点相同');
		多料盘管理输出.错误代码:=E_错误码.取料参考点错误不能和起始点相同;
	ELSE
		取料流程:=7;
	END_IF
END_IF

IF 取料流程=7 THEN
	//左上
		IF ST_料盘配置V1_xg_0[多料盘管理输入.料盘选择].x取料方位=0 THEN
			i行起始:=0;
			i行结束:=料盘配置[多料盘管理输入.料盘选择].行数-1;
			i列起始:=0;
			i列结束:=料盘配置[多料盘管理输入.料盘选择].列数-1;
			i行递增:=1;
			i列递增:=1;
		ELSIF ST_料盘配置V1_xg_0[多料盘管理输入.料盘选择].x取料方位=1 THEN
			i行起始:=0;
			i行结束:=料盘配置[多料盘管理输入.料盘选择].行数-1;
			i列起始:=料盘配置[多料盘管理输入.料盘选择].列数-1;
			i列结束:=0;
			i行递增:=1;
			i列递增:=-1;
		ELSIF ST_料盘配置V1_xg_0[多料盘管理输入.料盘选择].x取料方位=2 THEN
			i行起始:=料盘配置[多料盘管理输入.料盘选择].行数-1;
			i行结束:=0;
			i列起始:=0;
			i列结束:=料盘配置[多料盘管理输入.料盘选择].列数-1;
			i行递增:=-1;
			i列递增:=1;
		ELSIF ST_料盘配置V1_xg_0[多料盘管理输入.料盘选择].x取料方位=3 THEN
			i行起始:=料盘配置[多料盘管理输入.料盘选择].行数-1;
			i行结束:=0;
			i列起始:=料盘配置[多料盘管理输入.料盘选择].列数-1;
			i列结束:=0;
			i行递增:=-1;
			i列递增:=-1;
		END_IF
		取料流程:=10;
END_IF

IF 取料流程=10 THEN

	FOR i:=i行起始 TO i行结束 BY i行递增 DO
		FOR j:=i列起始 TO i列结束 BY i列递增 DO
			IF 多料盘管理数据.料盘管理数据[多料盘管理输入.料盘选择].屏蔽点位[i,j]=FALSE THEN
				IF 多料盘管理数据.料盘管理数据[多料盘管理输入.料盘选择].点位状态[i,j]=E_点位状态.有料 THEN
					临时定位行号:=i;
					临时定位列号:=j;
					取料流程:=12;
					EXIT;
				END_IF

				IF i=i行结束 AND j=i列结束 THEN
					多料盘管理输出.错误:=TRUE;
					报错料盘:=多料盘管理输入.料盘选择;
   					多料盘管理输出.错误信息 :=Standard.CONCAT(Standard.CONCAT('料盘', TO_STRING(多料盘管理输入.料盘选择)), '没料了');
					多料盘管理输出.错误代码:=E_错误码.料盘取料空料;
				END_IF
			END_IF
		END_FOR

		IF 取料流程<>10 THEN
			EXIT;
		END_IF
	END_FOR

END_IF

IF 取料流程=12 THEN
	料盘轴运动输入.x定位位置:=料盘轴运动输入.目标位置[0]:=多料盘管理输出.目标X位置 := 料盘配置[多料盘管理输入.料盘选择].起始X坐标 +
								临时定位列号 * 料盘配置[多料盘管理输入.料盘选择].列间距 * x取料方向X +
								料盘配置[多料盘管理输入.料盘选择].点位偏移[临时定位行号, 临时定位列号].x点位偏移;

	料盘轴运动输入.y定位位置:=料盘轴运动输入.目标位置[1]:=多料盘管理输出.目标Y位置 := 料盘配置[多料盘管理输入.料盘选择].起始Y坐标 +
								临时定位行号 * 料盘配置[多料盘管理输入.料盘选择].行间距 * x取料方向Y +
								料盘配置[多料盘管理输入.料盘选择].点位偏移[临时定位行号, 临时定位列号].y点位偏移;

	料盘轴运动输入.z定位位置:=多料盘管理输出.目标Z位置 := 料盘配置[多料盘管理输入.料盘选择].Z轴高度 +
								料盘配置[多料盘管理输入.料盘选择].点位偏移[临时定位行号, 临时定位列号].z点位偏移;

// 	料盘轴运动输入.xy插补速度:=多料盘管理配置.xy插补速度;
// 	料盘轴运动输入.xy插补加速度:=多料盘管理配置.xy插补加速度;
// 	料盘轴运动输入.xy插补减速度:=多料盘管理配置.xy插补减速度;

	料盘轴运动输入.x定位速度:=多料盘管理配置.x速度;
	料盘轴运动输入.x定位加速度:=多料盘管理配置.x加速度;
	料盘轴运动输入.x定位减速度:=多料盘管理配置.x减速度;

	料盘轴运动输入.y定位速度:=多料盘管理配置.y速度;
	料盘轴运动输入.y定位加速度:=多料盘管理配置.y加速度;
	料盘轴运动输入.y定位减速度:=多料盘管理配置.y减速度;

	IF 料盘工艺配置[多料盘管理输入.料盘选择].取料z轴下降减速动作.启用=1 THEN
		IF z轴.fActPosition>料盘工艺配置[多料盘管理输入.料盘选择].取料z轴下降减速动作.取料减速位置 THEN
			料盘轴运动输入.z定位速度:= 料盘工艺配置[多料盘管理输入.料盘选择].取料z轴下降减速动作.取料减速速度;
		ELSE
			料盘轴运动输入.z定位速度:=多料盘管理配置.z速度;
		END_IF
	ELSE
		料盘轴运动输入.z定位速度:=多料盘管理配置.z速度;
	END_IF

	料盘轴运动输入.z定位加速度:=多料盘管理配置.z加速度;
	料盘轴运动输入.z定位减速度:=多料盘管理配置.z减速度;

	IF x轴.nAxisState=Standstill  AND y轴.nAxisState=Standstill AND NOT 多料盘管理输入.暂停 THEN
		//料盘轴运动输入.插补启动:=TRUE;

		料盘轴运动输入.x轴定位:=TRUE;
		料盘轴运动输入.y轴定位:=TRUE;
		取料流程:=13;
	ELSIF 多料盘管理输入.暂停 THEN
		多料盘管理输出.暂停完成:=TRUE;
	END_IF
ELSIF 取料流程=13 THEN
	IF x轴.nAxisState=Standstill  AND y轴.nAxisState=Standstill AND NOT 多料盘管理输入.暂停 THEN
		//料盘轴运动输入.插补启动:=TRUE;

		料盘轴运动输入.x轴定位:=TRUE;
		料盘轴运动输入.y轴定位:=TRUE;
	//ELSIF 多料盘管理输入.暂停 THEN
	//	多料盘管理输出.暂停完成:=TRUE;
	END_IF
	IF 插补定位完成 AND x轴.nAxisState=Standstill  AND y轴.nAxisState=Standstill AND NOT 多料盘管理输入.暂停  THEN

		//料盘轴运动输入.插补启动:=FALSE;
		料盘轴运动输入.x轴定位:=FALSE;
		料盘轴运动输入.y轴定位:=FALSE;

		取料流程:=14;
	ELSIF 多料盘管理输入.暂停 THEN
		多料盘管理输出.暂停完成:=TRUE;

	END_IF
END_IF

IF 取料流程=14 THEN
	IF z轴定位到位=FALSE AND z轴.nAxisState=Standstill AND NOT 多料盘管理输入.暂停 THEN
			(* 移动轴 *)
			料盘轴运动输入.Z轴定位:=TRUE;
			取料流程:=14;
	ELSIF z轴定位到位 AND 多料盘管理输入.暂停 THEN
		多料盘管理输出.暂停完成:=TRUE;
	END_IF
	IF 料盘工艺配置[多料盘管理输入.料盘选择].取料z轴下降减速动作.启用=1 THEN
		IF z轴.fActPosition>料盘工艺配置[多料盘管理输入.料盘选择].取料z轴下降减速动作.取料减速位置 THEN
			料盘轴运动输入.z定位速度:= 料盘工艺配置[多料盘管理输入.料盘选择].取料z轴下降减速动作.取料减速速度;

		END_IF
	END_IF
	IF z轴定位到位 AND z轴.nAxisState=Standstill AND NOT 多料盘管理输入.暂停  THEN
		料盘轴运动输入.Z轴定位:=FALSE;

		IF 料盘工艺配置[多料盘管理输入.料盘选择].取料附加动作.模式 =0 THEN
			多料盘管理数据.料盘管理数据[多料盘管理输入.料盘选择].点位状态[临时定位行号,临时定位列号]:=E_点位状态.无料;
			多料盘管理输出.料盘运动状态:=E_料盘运动状态.待机;
			多料盘管理输出.到达定位位置:=TRUE;
			取料流程:=0;
		ELSIF 料盘工艺配置[多料盘管理输入.料盘选择].取料附加动作.模式 =1 THEN
			取料流程:=20;
		END_IF
	END_IF
ELSIF 取料流程=20 THEN
	IF 料盘工艺配置[多料盘管理输入.料盘选择].取料附加动作.索引=0 AND x轴.nAxisState=Standstill AND NOT 多料盘管理输入.暂停 THEN
		料盘轴运动输入.X定位位置:=多料盘管理输出.目标X位置 := 料盘工艺配置[多料盘管理输入.料盘选择].取料附加动作.偏移值+x轴.fActPosition;
		料盘轴运动输入.x定位速度:= 料盘工艺配置[多料盘管理输入.料盘选择].取料附加动作.速度;
		料盘轴运动输入.x定位加速度:= 料盘工艺配置[多料盘管理输入.料盘选择].取料附加动作.加速度;
		料盘轴运动输入.x定位减速度:=料盘工艺配置[多料盘管理输入.料盘选择].取料附加动作.减速度;
		料盘轴运动输入.x轴定位:=TRUE;
		取料流程:=30;
	ELSIF 料盘工艺配置[多料盘管理输入.料盘选择].取料附加动作.索引=1 AND y轴.nAxisState=Standstill AND NOT 多料盘管理输入.暂停 THEN
		料盘轴运动输入.y定位位置:=多料盘管理输出.目标y位置 := 料盘工艺配置[多料盘管理输入.料盘选择].取料附加动作.偏移值+y轴.fActPosition;
		料盘轴运动输入.y定位速度:=料盘工艺配置[多料盘管理输入.料盘选择].取料附加动作.速度;
		料盘轴运动输入.y定位加速度:=料盘工艺配置[多料盘管理输入.料盘选择].取料附加动作.加速度;
		料盘轴运动输入.y定位减速度:=料盘工艺配置[多料盘管理输入.料盘选择].取料附加动作.减速度;
		料盘轴运动输入.y轴定位:=TRUE;
		取料流程:=30;
	ELSIF 料盘工艺配置[多料盘管理输入.料盘选择].取料附加动作.索引=2 AND z轴.nAxisState=Standstill AND NOT 多料盘管理输入.暂停 THEN
		料盘轴运动输入.z定位位置:=多料盘管理输出.目标z位置 := 料盘工艺配置[多料盘管理输入.料盘选择].取料附加动作.偏移值+z轴.fActPosition;
		料盘轴运动输入.z定位速度:=料盘工艺配置[多料盘管理输入.料盘选择].取料附加动作.速度;
		料盘轴运动输入.z定位加速度:=料盘工艺配置[多料盘管理输入.料盘选择].取料附加动作.加速度;
		料盘轴运动输入.z定位减速度:=料盘工艺配置[多料盘管理输入.料盘选择].取料附加动作.减速度;
		料盘轴运动输入.z轴定位:=TRUE;
		取料流程:=30;
	ELSIF 多料盘管理输入.暂停 THEN
		多料盘管理输出.暂停完成:=TRUE;
	END_IF

ELSIF 取料流程=30 THEN
	IF 料盘工艺配置[多料盘管理输入.料盘选择].取料附加动作.索引=0 THEN
		IF x轴定位到位 AND x轴.nAxisState=Standstill THEN
			多料盘管理数据.料盘管理数据[多料盘管理输入.料盘选择].点位状态[临时定位行号,临时定位列号]:=E_点位状态.无料;
			料盘轴运动输入.x轴定位:=FALSE;
			多料盘管理输出.料盘运动状态:=E_料盘运动状态.待机;
			多料盘管理输出.到达定位位置:=TRUE;
			取料流程:=0;
		END_IF
	ELSIF 料盘工艺配置[多料盘管理输入.料盘选择].取料附加动作.索引=1 THEN
		IF y轴定位到位 AND y轴.nAxisState=Standstill THEN
			多料盘管理数据.料盘管理数据[多料盘管理输入.料盘选择].点位状态[临时定位行号,临时定位列号]:=E_点位状态.无料;
			料盘轴运动输入.y轴定位:=FALSE;
			多料盘管理输出.料盘运动状态:=E_料盘运动状态.待机;
			多料盘管理输出.到达定位位置:=TRUE;
			取料流程:=0;
		END_IF
	ELSIF 料盘工艺配置[多料盘管理输入.料盘选择].取料附加动作.索引=2 THEN
		IF z轴定位到位 AND z轴.nAxisState=Standstill THEN
			多料盘管理数据.料盘管理数据[多料盘管理输入.料盘选择].点位状态[临时定位行号,临时定位列号]:=E_点位状态.无料;
			料盘轴运动输入.z轴定位:=FALSE;
			多料盘管理输出.料盘运动状态:=E_料盘运动状态.待机;
			多料盘管理输出.到达定位位置:=TRUE;
			取料流程:=0;
		END_IF
	END_IF
END_IF

(* ---- FB_多料盘管理.ACT_自动放料.action.st ---- *)
放料上升沿(CLK:=多料盘管理输入.放料 AND 多料盘管理输入.手自动, Q=> );
放料完成上升沿(CLK:= 多料盘管理输入.放料完成 AND 多料盘管理输入.手自动, Q=> );

IF GVL_系统变量.全局状态=E_系统运行状态.系统状态_故障 THEN
	料盘轴运动输入.x轴定位:=FALSE;
	料盘轴运动输入.y轴定位:=FALSE;
	料盘轴运动输入.Z轴定位:=FALSE;
	料盘轴运动输入.插补启动:=FALSE;
	RETURN;
END_IF

IF GVL_系统变量.全局状态<>E_系统运行状态.系统状态_运行 AND GVL_系统变量.全局状态<>E_系统运行状态.系统状态_清料中  AND GVL_系统变量.全局状态<>E_系统运行状态.系统状态_暂停中 THEN

	RETURN;
END_IF

IF 放料完成上升沿.q THEN
	多料盘管理数据.料盘管理数据[多料盘管理输入.料盘选择].点位状态[临时定位行号,临时定位列号]:=E_点位状态.有料;
END_IF

IF 放料上升沿.Q AND 轴可运动 AND 流程可运行
	AND NOT 多料盘管理输入.到初始位 AND NOT 多料盘管理输入.取料 AND NOT 多料盘管理输入.定位
	 AND NOT 多料盘管理输入.暂停 AND NOT 多料盘管理输出.错误 AND
	(多料盘管理输出.料盘运动状态=E_料盘运动状态.待机
	OR 多料盘管理输出.料盘运动状态=E_料盘运动状态.暂停)
THEN
	料盘轴运动输入.x轴定位:=FALSE;
	料盘轴运动输入.y轴定位:=FALSE;
	料盘轴运动输入.Z轴定位:=FALSE;
	料盘轴运动输入.插补启动:=FALSE;
	多料盘管理输出.到达定位位置:=FALSE;
	IF 多料盘管理输出.料盘运动状态=E_料盘运动状态.暂停 THEN
		多料盘管理输出.料盘运动状态:=E_料盘运动状态.到放料位中;
		放料流程:=12;
	ELSE
		多料盘管理输出.料盘运动状态:=E_料盘运动状态.到放料位中;
		放料流程:=2;
	END_IF

ELSE
	;
END_IF;

IF 放料流程=2 THEN
	IF z轴在待料位=FALSE THEN
		料盘轴运动输入.z定位位置:=多料盘管理输出.目标Z位置 := 多料盘管理配置.z轴待料位;
		料盘轴运动输入.z定位速度:=多料盘管理配置.z速度;
		料盘轴运动输入.z定位加速度:=多料盘管理配置.z加速度;
		料盘轴运动输入.z定位减速度:=多料盘管理配置.z减速度;
		料盘轴运动输入.Z轴定位:=TRUE;
		放料流程:=5;
	ELSE
		放料流程:=5;
	END_IF
END_IF

IF 放料流程=5 THEN
	IF z轴在待料位=FALSE AND NOT 多料盘管理输入.暂停 THEN
		料盘轴运动输入.z定位位置:=多料盘管理输出.目标Z位置 := 多料盘管理配置.z轴待料位;
		料盘轴运动输入.z定位速度:=多料盘管理配置.z速度;
		料盘轴运动输入.z定位加速度:=多料盘管理配置.z加速度;
		料盘轴运动输入.z定位减速度:=多料盘管理配置.z减速度;
		料盘轴运动输入.Z轴定位:=TRUE;
	END_IF
	IF z轴在待料位 AND z轴.nAxisState=Standstill AND NOT 多料盘管理输入.暂停  THEN
		料盘轴运动输入.Z轴定位:=FALSE;
		放料流程:=6;
	ELSIF 多料盘管理输入.暂停 THEN
		多料盘管理输出.暂停完成:=TRUE;
	END_IF
END_IF

IF 放料流程=6 THEN
	IF FC_方向判断(
	i方向X:= x放料方向X,
	i方向Y:= x放料方向Y ,
	f起始点X:=料盘配置[多料盘管理输入.料盘选择].放料起始X坐标 ,
	f起始点Y:= 料盘配置[多料盘管理输入.料盘选择].放料起始Y坐标 ,
	f参考点X:=ST_料盘配置V1_xg_0[多料盘管理输入.料盘选择].lf放料参考点x坐标 ,
	f参考点Y:=ST_料盘配置V1_xg_0[多料盘管理输入.料盘选择].lf放料参考点y坐标 )=1 THEN
		多料盘管理输出.错误:=TRUE;
		报错料盘:=多料盘管理输入.料盘选择;
		多料盘管理输出.错误信息 :=Standard.CONCAT(Standard.CONCAT('料盘', TO_STRING(多料盘管理输入.料盘选择)), '放料参考点错误,不能和起始点相同');
		多料盘管理输出.错误代码:=E_错误码.放料参考点错误不能和起始点相同;
	ELSE
		放料流程:=7;
	END_IF
END_IF

IF 放料流程=7 THEN
	//左上
		IF ST_料盘配置V1_xg_0[多料盘管理输入.料盘选择].x放料方位=0 THEN
			i行起始:=0;
			i行结束:=料盘配置[多料盘管理输入.料盘选择].行数-1;
			i列起始:=0;
			i列结束:=料盘配置[多料盘管理输入.料盘选择].列数-1;
			i行递增:=1;
			i列递增:=1;
		ELSIF ST_料盘配置V1_xg_0[多料盘管理输入.料盘选择].x放料方位=1 THEN
			i行起始:=0;
			i行结束:=料盘配置[多料盘管理输入.料盘选择].行数-1;
			i列起始:=料盘配置[多料盘管理输入.料盘选择].列数-1;
			i列结束:=0;
			i行递增:=1;
			i列递增:=-1;
		ELSIF ST_料盘配置V1_xg_0[多料盘管理输入.料盘选择].x放料方位=2 THEN
			i行起始:=料盘配置[多料盘管理输入.料盘选择].行数-1;
			i行结束:=0;
			i列起始:=0;
			i列结束:=料盘配置[多料盘管理输入.料盘选择].列数-1;
			i行递增:=-1;
			i列递增:=1;
		ELSIF ST_料盘配置V1_xg_0[多料盘管理输入.料盘选择].x放料方位=3 THEN
			i行起始:=料盘配置[多料盘管理输入.料盘选择].行数-1;
			i行结束:=0;
			i列起始:=料盘配置[多料盘管理输入.料盘选择].列数-1;
			i列结束:=0;
			i行递增:=-1;
			i列递增:=-1;
		END_IF
		放料流程:=10;
END_IF

IF 放料流程=10 THEN

	FOR i:=i行起始 TO i行结束 BY i行递增 DO
		FOR j:=i列起始 TO i列结束 BY i列递增 DO
			IF 多料盘管理数据.料盘管理数据[多料盘管理输入.料盘选择].屏蔽点位[i,j]=FALSE THEN

				IF 多料盘管理数据.料盘管理数据[多料盘管理输入.料盘选择].点位状态[i,j]=E_点位状态.无料 THEN
					临时定位行号:=i;
					临时定位列号:=j;
					放料流程:=12;
					EXIT;
				END_IF

				IF i=i行结束 AND j=i列结束 THEN
					多料盘管理输出.错误:=TRUE;
					报错料盘:=多料盘管理输入.料盘选择;
   					多料盘管理输出.错误信息 :=Standard.CONCAT(Standard.CONCAT('料盘', TO_STRING(多料盘管理输入.料盘选择)), '料满了');
					多料盘管理输出.错误代码:=E_错误码.料盘放料满料;
				END_IF
			END_IF
		END_FOR

		IF 放料流程<>10 THEN
			EXIT;
		END_IF
	END_FOR
END_IF

IF 放料流程=12 THEN
	料盘轴运动输入.x定位位置:=料盘轴运动输入.目标位置[0]:=多料盘管理输出.目标X位置 := 料盘配置[多料盘管理输入.料盘选择].放料起始X坐标 +
								临时定位列号 * 料盘配置[多料盘管理输入.料盘选择].列间距 *x放料方向X +
								料盘配置[多料盘管理输入.料盘选择].点位偏移[临时定位行号, 临时定位列号].x点位偏移;

	料盘轴运动输入.y定位位置:=料盘轴运动输入.目标位置[1]:=多料盘管理输出.目标Y位置 := 料盘配置[多料盘管理输入.料盘选择].放料起始Y坐标 +
								临时定位行号 * 料盘配置[多料盘管理输入.料盘选择].行间距 *x放料方向Y +
								料盘配置[多料盘管理输入.料盘选择].点位偏移[临时定位行号, 临时定位列号].y点位偏移;

	料盘轴运动输入.z定位位置:=多料盘管理输出.目标Z位置 := 料盘配置[多料盘管理输入.料盘选择].放料Z轴高度 +
								料盘配置[多料盘管理输入.料盘选择].点位偏移[临时定位行号, 临时定位列号].z点位偏移;

// 	料盘轴运动输入.xy插补速度:=多料盘管理配置.xy插补速度;
// 	料盘轴运动输入.xy插补加速度:=多料盘管理配置.xy插补加速度;
// 	料盘轴运动输入.xy插补减速度:=多料盘管理配置.xy插补减速度;

	料盘轴运动输入.x定位速度:=多料盘管理配置.x速度;
	料盘轴运动输入.x定位加速度:=多料盘管理配置.x加速度;
	料盘轴运动输入.x定位减速度:=多料盘管理配置.x减速度;

	料盘轴运动输入.y定位速度:=多料盘管理配置.y速度;
	料盘轴运动输入.y定位加速度:=多料盘管理配置.y加速度;
	料盘轴运动输入.y定位减速度:=多料盘管理配置.y减速度;

	IF 料盘工艺配置[多料盘管理输入.料盘选择].放料z轴下降减速动作.启用=1 THEN
		IF z轴.fActPosition>料盘工艺配置[多料盘管理输入.料盘选择].放料z轴下降减速动作.放料减速位置 THEN
			料盘轴运动输入.z定位速度:= 料盘工艺配置[多料盘管理输入.料盘选择].放料z轴下降减速动作.放料减速速度;
		ELSE
			料盘轴运动输入.z定位速度:=多料盘管理配置.z速度;
		END_IF
	ELSE
		料盘轴运动输入.z定位速度:=多料盘管理配置.z速度;
	END_IF
	料盘轴运动输入.z定位加速度:=多料盘管理配置.z加速度;
	料盘轴运动输入.z定位减速度:=多料盘管理配置.z减速度;

	IF x轴.nAxisState=Standstill  AND y轴.nAxisState=Standstill AND NOT 多料盘管理输入.暂停 THEN
		//料盘轴运动输入.插补启动:=TRUE;
		料盘轴运动输入.x轴定位:=TRUE;
		料盘轴运动输入.y轴定位:=TRUE;
		放料流程:=13;
	ELSIF 多料盘管理输入.暂停 THEN
		多料盘管理输出.暂停完成:=TRUE;
	END_IF

ELSIF 放料流程=13 THEN
	IF x轴.nAxisState=Standstill  AND y轴.nAxisState=Standstill AND NOT 多料盘管理输入.暂停 THEN
		//料盘轴运动输入.插补启动:=TRUE;

		料盘轴运动输入.x轴定位:=TRUE;
		料盘轴运动输入.y轴定位:=TRUE;
	//ELSIF 多料盘管理输入.暂停 THEN
	//	多料盘管理输出.暂停完成:=TRUE;
	END_IF
	IF 插补定位完成 AND x轴.nAxisState=Standstill  AND y轴.nAxisState=Standstill AND NOT 多料盘管理输入.暂停  THEN

		//料盘轴运动输入.插补启动:=FALSE;
		料盘轴运动输入.x轴定位:=FALSE;
		料盘轴运动输入.y轴定位:=FALSE;

		放料流程:=14;
	ELSIF 多料盘管理输入.暂停 THEN
		多料盘管理输出.暂停完成:=TRUE;

	END_IF
END_IF

IF 放料流程=14 THEN
	IF z轴定位到位=FALSE AND z轴.nAxisState=Standstill AND NOT 多料盘管理输入.暂停  THEN
			料盘轴运动输入.Z轴定位:=TRUE;
		ELSIF z轴定位到位 AND 多料盘管理输入.暂停 THEN
			多料盘管理输出.暂停完成:=TRUE;
		END_IF
	IF 料盘工艺配置[多料盘管理输入.料盘选择].放料z轴下降减速动作.启用=1 THEN
		IF z轴.fActPosition>料盘工艺配置[多料盘管理输入.料盘选择].放料z轴下降减速动作.放料减速位置 THEN
			料盘轴运动输入.z定位速度:= 料盘工艺配置[多料盘管理输入.料盘选择].放料z轴下降减速动作.放料减速速度;

		END_IF

	END_IF

	IF z轴定位到位 AND z轴.nAxisState=Standstill AND NOT 多料盘管理输入.暂停  THEN
		料盘轴运动输入.Z轴定位:=FALSE;

		IF 料盘工艺配置[多料盘管理输入.料盘选择].放料附加动作.模式 =0 THEN
			多料盘管理数据.料盘管理数据[多料盘管理输入.料盘选择].点位状态[临时定位行号,临时定位列号]:=E_点位状态.有料;
			多料盘管理输出.料盘运动状态:=E_料盘运动状态.待机;
			多料盘管理输出.到达定位位置:=TRUE;
			放料流程:=0;
		ELSIF 料盘工艺配置[多料盘管理输入.料盘选择].放料附加动作.模式 =1 THEN
			放料流程:=20;
		END_IF
	END_IF
ELSIF 放料流程=20 THEN
	IF 料盘工艺配置[多料盘管理输入.料盘选择].放料附加动作.索引=0 AND x轴.nAxisState=Standstill AND NOT 多料盘管理输入.暂停 THEN
		料盘轴运动输入.X定位位置:=多料盘管理输出.目标X位置 := 料盘工艺配置[多料盘管理输入.料盘选择].放料附加动作.偏移值+x轴.fActPosition;
		料盘轴运动输入.x定位速度:= 料盘工艺配置[多料盘管理输入.料盘选择].放料附加动作.速度;
		料盘轴运动输入.x定位加速度:= 料盘工艺配置[多料盘管理输入.料盘选择].放料附加动作.加速度;
		料盘轴运动输入.x定位减速度:=料盘工艺配置[多料盘管理输入.料盘选择].放料附加动作.减速度;
		料盘轴运动输入.x轴定位:=TRUE;
		放料流程:=30;
	ELSIF 料盘工艺配置[多料盘管理输入.料盘选择].放料附加动作.索引=1 AND y轴.nAxisState=Standstill AND NOT 多料盘管理输入.暂停  THEN
		料盘轴运动输入.y定位位置:=多料盘管理输出.目标y位置 := 料盘工艺配置[多料盘管理输入.料盘选择].放料附加动作.偏移值+y轴.fActPosition;
		料盘轴运动输入.y定位速度:=料盘工艺配置[多料盘管理输入.料盘选择].放料附加动作.速度;
		料盘轴运动输入.y定位加速度:=料盘工艺配置[多料盘管理输入.料盘选择].放料附加动作.加速度;
		料盘轴运动输入.y定位减速度:=料盘工艺配置[多料盘管理输入.料盘选择].放料附加动作.减速度;
		料盘轴运动输入.y轴定位:=TRUE;
		放料流程:=30;
	ELSIF 料盘工艺配置[多料盘管理输入.料盘选择].放料附加动作.索引=2 AND z轴.nAxisState=Standstill AND NOT 多料盘管理输入.暂停  THEN
		料盘轴运动输入.z定位位置:=多料盘管理输出.目标z位置 := 料盘工艺配置[多料盘管理输入.料盘选择].放料附加动作.偏移值+z轴.fActPosition;
		料盘轴运动输入.z定位速度:=料盘工艺配置[多料盘管理输入.料盘选择].放料附加动作.速度;
		料盘轴运动输入.z定位加速度:=料盘工艺配置[多料盘管理输入.料盘选择].放料附加动作.加速度;
		料盘轴运动输入.z定位减速度:=料盘工艺配置[多料盘管理输入.料盘选择].放料附加动作.减速度;
		料盘轴运动输入.z轴定位:=TRUE;
		放料流程:=30;
	ELSIF 多料盘管理输入.暂停 THEN
		多料盘管理输出.暂停完成:=TRUE;
	END_IF

ELSIF 放料流程=30 THEN
	IF 料盘工艺配置[多料盘管理输入.料盘选择].放料附加动作.索引=0 THEN
		IF x轴定位到位 AND x轴.nAxisState=Standstill THEN
			多料盘管理数据.料盘管理数据[多料盘管理输入.料盘选择].点位状态[临时定位行号,临时定位列号]:=E_点位状态.有料;
			料盘轴运动输入.x轴定位:=FALSE;
			多料盘管理输出.料盘运动状态:=E_料盘运动状态.待机;
			多料盘管理输出.到达定位位置:=TRUE;
			放料流程:=0;
		END_IF
	ELSIF 料盘工艺配置[多料盘管理输入.料盘选择].放料附加动作.索引=1 THEN
		IF y轴定位到位 AND y轴.nAxisState=Standstill  THEN
			多料盘管理数据.料盘管理数据[多料盘管理输入.料盘选择].点位状态[临时定位行号,临时定位列号]:=E_点位状态.有料;
			料盘轴运动输入.y轴定位:=FALSE;
			多料盘管理输出.料盘运动状态:=E_料盘运动状态.待机;
			多料盘管理输出.到达定位位置:=TRUE;
			放料流程:=0;
		END_IF
	ELSIF 料盘工艺配置[多料盘管理输入.料盘选择].放料附加动作.索引=2 THEN
		IF z轴定位到位 AND z轴.nAxisState=Standstill THEN
			多料盘管理数据.料盘管理数据[多料盘管理输入.料盘选择].点位状态[临时定位行号,临时定位列号]:=E_点位状态.有料;
			料盘轴运动输入.z轴定位:=FALSE;
			多料盘管理输出.料盘运动状态:=E_料盘运动状态.待机;
			多料盘管理输出.到达定位位置:=TRUE;
			放料流程:=0;
		END_IF
	END_IF
END_IF

(* ---- FB_多料盘管理.ACT_自动状态控制.action.st ---- *)
//读取轴状态功能块
x轴状态(Axis:= x轴, Enable:=x轴.wCommunicationState=100);
y轴状态(Axis:= y轴, Enable:=y轴.wCommunicationState=100);
z轴状态(Axis:= z轴, Enable:=z轴.wCommunicationState=100);

手动急停上升沿(CLK:=多料盘管理输入HMI.急停 AND NOT 多料盘管理输入.手自动 , Q=> );

IF 手动急停上升沿.Q THEN
	放料流程:=0;
	取料流程:=0;
	定位流程:=0;
	手动定位流程:=0;
	指定取料流程:=0;
	指定放料流程:=0;
	手动取料流程:=0;
	手动放料流程:=0;
	多料盘管理输出.料盘运动状态:=E_料盘运动状态.待机;
	料盘轴运动输入.x轴定位:=FALSE;
	料盘轴运动输入.y轴定位:=FALSE;
	料盘轴运动输入.Z轴定位:=FALSE;
	料盘轴运动输入.插补启动:=FALSE;
	多料盘管理输出.错误:=FALSE;
    多料盘管理输出.错误信息 :='';
END_IF

IF 多料盘管理输入HMI.急停 THEN
	IF (FC_误差判断(实际值:=x轴.fActVelocity , 判断值:= 0, 误差值:=0.000001 )=FALSE OR
		FC_误差判断(实际值:=y轴.fActVelocity , 判断值:= 0, 误差值:=0.000001 )=FALSE)
		AND x轴状态.SynchronizedMotion AND y轴状态.SynchronizedMotion THEN
		料盘轴运动输入.插补停止:=TRUE;
	END_IF
	IF FC_误差判断(实际值:=x轴.fActVelocity , 判断值:= 0, 误差值:=0.000001 )=FALSE
		AND (x轴状态.DiscreteMotion OR x轴状态.ContinuousMotion) THEN
		料盘轴运动输入.x轴停止:=TRUE;
	END_IF
	IF FC_误差判断(实际值:=y轴.fActVelocity , 判断值:= 0, 误差值:=0.000001 )=FALSE
		AND (y轴状态.DiscreteMotion OR y轴状态.ContinuousMotion) THEN
		料盘轴运动输入.y轴停止:=TRUE;
	END_IF
	IF FC_误差判断(实际值:=z轴.fActVelocity , 判断值:= 0, 误差值:=0.000001 )=FALSE
		AND (z轴状态.DiscreteMotion OR z轴状态.ContinuousMotion) THEN
		料盘轴运动输入.z轴停止:=TRUE;
	END_IF
END_IF

急停上升沿(CLK:= 多料盘管理输入.急停, Q=> );

IF 急停上升沿.Q THEN
	放料流程:=0;
	取料流程:=0;
	定位流程:=0;
	手动定位流程:=0;
	指定取料流程:=0;
	指定放料流程:=0;
	手动取料流程:=0;
	手动放料流程:=0;
	多料盘管理输出.料盘运动状态:=E_料盘运动状态.待机;
	料盘轴运动输入.x轴定位:=FALSE;
	料盘轴运动输入.y轴定位:=FALSE;
	料盘轴运动输入.Z轴定位:=FALSE;
	料盘轴运动输入.插补启动:=FALSE;
	多料盘管理输出.错误:=FALSE;
    多料盘管理输出.错误信息 :='';
END_IF

IF 多料盘管理输入.急停 THEN
	IF (FC_误差判断(实际值:=x轴.fActVelocity , 判断值:= 0, 误差值:=0.000001 )=FALSE OR
		FC_误差判断(实际值:=y轴.fActVelocity , 判断值:= 0, 误差值:=0.000001 )=FALSE)
		AND x轴状态.SynchronizedMotion AND y轴状态.SynchronizedMotion THEN
		料盘轴运动输入.插补停止:=TRUE;
	END_IF
	IF FC_误差判断(实际值:=x轴.fActVelocity , 判断值:= 0, 误差值:=0.000001 )=FALSE
		AND (x轴状态.DiscreteMotion OR x轴状态.ContinuousMotion) THEN
		料盘轴运动输入.x轴停止:=TRUE;
	END_IF
	IF FC_误差判断(实际值:=y轴.fActVelocity , 判断值:= 0, 误差值:=0.000001 )=FALSE
		AND (y轴状态.DiscreteMotion OR y轴状态.ContinuousMotion) THEN
		料盘轴运动输入.y轴停止:=TRUE;
	END_IF
	IF FC_误差判断(实际值:=z轴.fActVelocity , 判断值:= 0, 误差值:=0.000001 )=FALSE
		AND (z轴状态.DiscreteMotion OR z轴状态.ContinuousMotion) THEN
		料盘轴运动输入.z轴停止:=TRUE;
	END_IF
END_IF

复位上升沿(CLK:=多料盘管理输入.复位 , Q=> );
IF  复位上升沿.Q THEN
	放料流程:=0;
	取料流程:=0;
	定位流程:=0;
	手动定位流程:=0;
	指定取料流程:=0;
	指定放料流程:=0;
	手动取料流程:=0;
	手动放料流程:=0;
	多料盘管理输出.料盘运动状态:=E_料盘运动状态.待机;
	料盘轴运动输入.x轴定位:=FALSE;
	料盘轴运动输入.y轴定位:=FALSE;
	料盘轴运动输入.Z轴定位:=FALSE;
	料盘轴运动输入.插补启动:=FALSE;
	多料盘管理输出.错误:=FALSE;
    多料盘管理输出.错误信息 :='';
END_IF
//复位块状态,加停止轴
IF 多料盘管理输入.复位  THEN

	IF (FC_误差判断(实际值:=x轴.fActVelocity , 判断值:= 0, 误差值:=0.000001 )=FALSE OR
		FC_误差判断(实际值:=y轴.fActVelocity , 判断值:= 0, 误差值:=0.000001 )=FALSE)
		AND x轴状态.SynchronizedMotion AND y轴状态.SynchronizedMotion THEN
		料盘轴运动输入.插补停止:=TRUE;
	END_IF
	IF FC_误差判断(实际值:=x轴.fActVelocity , 判断值:= 0, 误差值:=0.000001 )=FALSE
		AND (x轴状态.DiscreteMotion OR x轴状态.ContinuousMotion) THEN
		料盘轴运动输入.x轴停止:=TRUE;
	END_IF
	IF FC_误差判断(实际值:=y轴.fActVelocity , 判断值:= 0, 误差值:=0.000001 )=FALSE
		AND (y轴状态.DiscreteMotion OR y轴状态.ContinuousMotion) THEN
		料盘轴运动输入.y轴停止:=TRUE;
	END_IF
	IF FC_误差判断(实际值:=z轴.fActVelocity , 判断值:= 0, 误差值:=0.000001 )=FALSE
		AND (z轴状态.DiscreteMotion OR z轴状态.ContinuousMotion) THEN
		料盘轴运动输入.z轴停止:=TRUE;
	END_IF

ELSE
	多料盘管理输出.复位完成:=FALSE;
END_IF

// 暂停上升沿(CLK:=多料盘管理输入.暂停 , Q=> );
// IF 暂停上升沿.Q THEN
//
//
// 	IF (多料盘管理输出.料盘运动状态=E_料盘运动状态.到取料位中 OR 多料盘管理输出.料盘运动状态=E_料盘运动状态.到放料位中)
// 	AND (取料流程>=12 OR 放料流程>=12) THEN
// 		多料盘管理输出.料盘运动状态:=E_料盘运动状态.暂停;
// 	ELSE
// 		多料盘管理输出.料盘运动状态:=E_料盘运动状态.待机;
// 	END_IF
//
// 	放料流程:=0;
// 	取料流程:=0;
// 	定位流程:=0;
// 	手动定位流程:=0;
// 	料盘轴运动输入.x轴定位:=FALSE;
// 	料盘轴运动输入.y轴定位:=FALSE;
// 	料盘轴运动输入.Z轴定位:=FALSE;
// 	料盘轴运动输入.插补启动:=FALSE;
// END_IF

//暂停动作
IF NOT 多料盘管理输入.暂停 THEN
	多料盘管理输出.暂停完成:=FALSE;
END_IF
IF 多料盘管理输出.暂停完成  THEN
	料盘轴运动输入.x轴定位:=FALSE;
		料盘轴运动输入.y轴定位:=FALSE;
		料盘轴运动输入.Z轴定位:=FALSE;
		料盘轴运动输入.插补启动:=FALSE;
END_IF
// IF 多料盘管理输入.暂停  THEN
// 	IF (FC_误差判断(实际值:=x轴.fActVelocity , 判断值:= 0, 误差值:=0.000001 )=FALSE OR
// 		FC_误差判断(实际值:=y轴.fActVelocity , 判断值:= 0, 误差值:=0.000001 )=FALSE)
// 		AND x轴状态.SynchronizedMotion AND y轴状态.SynchronizedMotion THEN
// 		料盘轴运动输入.插补停止:=TRUE;
// 	END_IF
// 	IF FC_误差判断(实际值:=x轴.fActVelocity , 判断值:= 0, 误差值:=0.000001 )=FALSE
// 		AND (x轴状态.DiscreteMotion OR x轴状态.ContinuousMotion) THEN
// 		料盘轴运动输入.x轴停止:=TRUE;
// 	END_IF
// 	IF FC_误差判断(实际值:=y轴.fActVelocity , 判断值:= 0, 误差值:=0.000001 )=FALSE
// 		AND (y轴状态.DiscreteMotion OR y轴状态.ContinuousMotion) THEN
// 		料盘轴运动输入.y轴停止:=TRUE;
// 	END_IF
// 	IF FC_误差判断(实际值:=z轴.fActVelocity , 判断值:= 0, 误差值:=0.000001 )=FALSE
// 		AND (z轴状态.DiscreteMotion OR z轴状态.ContinuousMotion) THEN
// 		料盘轴运动输入.z轴停止:=TRUE;
// 	END_IF
//
//
// ELSE
// 	多料盘管理输出.暂停完成:=FALSE;
// END_IF

IF FC_误差判断(实际值:=x轴.fActVelocity , 判断值:= 0, 误差值:=0.000001 ) AND
		FC_误差判断(实际值:=y轴.fActVelocity , 判断值:= 0, 误差值:=0.000001 ) AND
		FC_误差判断(实际值:=z轴.fActVelocity , 判断值:= 0, 误差值:=0.000001 ) THEN
		料盘轴运动输入.插补停止:=FALSE;
		料盘轴运动输入.x轴停止:=FALSE;
		料盘轴运动输入.y轴停止:=FALSE;
		料盘轴运动输入.z轴停止:=FALSE;

		IF 多料盘管理输入.暂停 THEN
			多料盘管理输出.暂停完成:=TRUE;
		END_IF
		IF 多料盘管理输入.复位 THEN
			多料盘管理输出.复位完成:=TRUE;
		END_IF
	END_IF

IF NOT x轴状态.Standstill OR NOT y轴状态.Standstill OR NOT z轴状态.Standstill THEN
	FOR i:=0 TO 4 BY 1 DO
		多料盘管理输出.定位号定位到位[i]:=FALSE;
		多料盘管理输出.到达定位位置:=FALSE;
	END_FOR

END_IF

多料盘管理输出.移动X轴信号:=x轴状态.DiscreteMotion OR x轴状态.ContinuousMotion;
多料盘管理输出.移动y轴信号:=y轴状态.DiscreteMotion OR y轴状态.ContinuousMotion;
多料盘管理输出.移动z轴信号:=z轴状态.DiscreteMotion OR z轴状态.ContinuousMotion;
